(* CoDeSys 2.3 project: cy-wg-03_013.pro *)
(* Title: ClevergyAS - SanFelice *)
(* Version: 0.0 *)
(* Author: Andrea Ravasio *)
(* Libraries: serial_interface_01.lib 22.4.13 11:50:14, SerComm.lib 31.5.11 07:54:36, MBus_03.lib 9.2.13 16:51:58, Util.lib 18.5.10 14:14:28, Visual.lib 2.12.10 13:48:34, WagoLibIdent.lib 25.2.13 10:12:16, WagoLibStatus.lib 2.12.10 13:48:32, SysLibFile.lib 2.12.10 13:48:34, SysLibRtc.lib 2.12.10 13:48:32, SysLibSockets.lib 10.2.11 08:20:54, SysLibEvent.lib 2.12.10 13:48:34, SysLibPlcCtrl.lib 2.12.10 13:48:32, Standard.lib 2.12.10 13:48:34, SYSLIBCALLBACK.LIB 2.12.10 13:48:32 *)

(* PLC configuration (modules and I/O channels)
0750-0402 4 DI 24 V DC 3.0ms [Type_1_4_Channels] node 0, in %IB24 out %QB4 {INTTypePAAssignment = PLC; INTTypeModule = plugged}
  VPN_ST2 AT %IX12.0 [BOOLOnX_I] Ch_1 Digital input
  KEY_QE_ST AT %IX12.1 [BOOLOnX_I] Ch_2 Digital input
  AT %IX12.2 [BOOLOnX_I] Ch_3 Digital input
  PORT01_DI AT %IX12.3 [BOOLOnX_I] Ch_4 Digital input
0750-0402 4 DI 24 V DC 3.0ms [Type_1_4_Channels] node 1, in %IB24 out %QB4 {INTTypePAAssignment = PLC; INTTypeModule = plugged}
  GAS02_DI AT %IX12.4 [BOOLOnX_I] Ch_1 Digital input
  GAS01_DI AT %IX12.5 [BOOLOnX_I] Ch_2 Digital input
  AT %IX12.6 [BOOLOnX_I] Ch_3 Digital input
  AT %IX12.7 [BOOLOnX_I] Ch_4 Digital input
0750-0504 4 DO 24V DC 0.5A [Type_10_4_Channels] node 2, in %IX12.4 out %QB4 {INTTypePAAssignment = PLC; INTTypeModule = plugged}
  AT %QX2.0 [BOOLOnX_Q] Ch_1 Digital output
  AT %QX2.1 [BOOLOnX_Q] Ch_2 Digital output
  AT %QX2.2 [BOOLOnX_Q] Ch_3 Digital output
  AT %QX2.3 [BOOLOnX_Q] Ch_4 Digital output
0750-0504 4 DO 24V DC 0.5A [Type_10_4_Channels] node 3, in %IB25 out %QB4 {INTTypePAAssignment = PLC; INTTypeModule = plugged}
  AT %QX2.4 [BOOLOnX_Q] Ch_1 Digital output
  AT %QX2.5 [BOOLOnX_Q] Ch_2 Digital output
  TEST1 AT %QX2.6 [BOOLOnX_Q] Ch_3 Digital output
  TEST2 AT %QX2.7 [BOOLOnX_Q] Ch_4 Digital output
0750-0464#02 2/4 AI RTD / ADJ./ HA [Type_44_2_Channels] node 4, in %IB20 out %QB0 {INTTypePAAssignment = PLC; INTTypeModule = plugged}
  TT_S01 AT %IW0 [INTOnW_I] Ch_1 signed Input value
  AT %IW1 [INTOnW_I] Ch_2 signed Input value
0750-0472 2 AI 0-20mA 16 Bit S.E. [Type_8_2_Channels] node 5, in %IB20 out %QB0 {INTTypePAAssignment = PLC; INTTypeModule = plugged}
  TT_S07 AT %IW2 [WORDOnW_I] I 1: Analog Input
  TT_S06 AT %IW3 [WORDOnW_I] I 2: Analog Input
0750-0472 2 AI 0-20mA 16 Bit S.E. [Type_8_2_Channels] node 6, in %IB24 out %QB0 {INTTypePAAssignment = PLC; INTTypeModule = plugged}
  TT_S05 AT %IW4 [WORDOnW_I] I 1: Analog Input
  TT_S04 AT %IW5 [WORDOnW_I] I 2: Analog Input
0750-0472 2 AI 0-20mA 16 Bit S.E. [Type_8_2_Channels] node 7, in %IB28 out %QB0 {INTTypePAAssignment = PLC; INTTypeModule = plugged}
  TT_S03 AT %IW6 [WORDOnW_I] I 1: Analog Input
  TT_S02 AT %IW7 [WORDOnW_I] I 2: Analog Input
0750-0472 2 AI 0-20mA 16 Bit S.E. [Type_8_2_Channels] node 8, in %IB32 out %QB0 {INTTypePAAssignment = PLC; INTTypeModule = plugged}
  PORT01_AI AT %IW8 [WORDOnW_I] I 1: Analog Input
  AT %IW9 [WORDOnW_I] I 2: Analog Input
0750-0650/0003-0000#03 RS 232 C Interface (Adjustable), 3 Byte [Type_21_1_Channels] node 9, in %IB36 out %QB0 {INTTypePAAssignment = PLC; INTTypeModule = plugged}
  AT %IX10.0 [BOOLOnX_I] Transmission acknowledgement
  AT %IX10.1 [BOOLOnX_I] Reception request
  AT %IX10.2 [BOOLOnX_I] Initialization acknowledgement
  AT %IX10.3 [BOOLOnX_I] Input buffer is full
  AT %IX10.4 [BOOLOnX_I] Number of received characters Bit 0
  AT %IX10.5 [BOOLOnX_I] Number of received characters Bit 1
  AT %IX10.6 [BOOLOnX_I] Number of received characters Bit 2
  AT %IB21 [BYTEOnB_I] Input data Byte 0
  AT %IB22 [BYTEOnB_I] Input data Byte 1
  AT %IB23 [BYTEOnB_I] Input data Byte 2
  AT %QX0.0 [BOOLOnX_Q] Transmission request
  AT %QX0.1 [BOOLOnX_Q] Reception acknowledgement
  AT %QX0.2 [BOOLOnX_Q] Initialization request
  AT %QX0.4 [BOOLOnX_Q] Number of characters Bit 0
  AT %QX0.5 [BOOLOnX_Q] Number of characters Bit 1
  AT %QX0.6 [BOOLOnX_Q] Number of characters Bit 2
  AT %QB1 [BYTEOnB_Q] Output data Byte 0
  AT %QB2 [BYTEOnB_Q] Output data Byte 1
  AT %QB3 [BYTEOnB_Q] Output data Byte 2
Fieldbus variables [FB_VARS] node 1, in %IB0 out %QB0
Flag variables [FLAG_VARS] node 2, in %IB0 out %QB0
Modbus-Master [MB_MASTER] node 3, in %IB0 out %QB0
*)

(* Global variable list: Global_Constants *)
VAR_GLOBAL CONSTANT

	Plant_NAME			: STRING :='cySN:3 cyVER:14 - San Felice';
	Plant_SN			: DWORD :=3;   		(* S/N Impianto di telecontrollo *)
	Plant_SW_VER		: WORD  :=14;		(* Versione SW installata *)

	(* Parameters *)
	Plant_DefaultTAmb	: INT	:=100;		(* [.1°C] Temperatura ambiente di default in caso di rottura sonda *)

	(* Filesystem *)
	FilesPath  			: STRING :='S:\';

	(* TCP Logger *)
	Logger_SERVER		: STRING:='';
	Logger_IP			: STRING:='192.168.100.3';
	Logger_PORT			: WORD  :=80;
	Logger_GETSTART		: STRING:='GET /cygmsrv/hsgm.ashx?';
	Logger_GETEND		: STRING:='$R$N$R$N';
	Logger_CHECK		: STRING:='True';
	Logger_CRLF			: STRING:='$R$N';
	Logger_DataFile		: STRING:='S:\LOG.DAT';
	Logger_DataFileOld	: STRING:='S:\LOG.BCK';
	Logger_IndexFile	: STRING:='S:\LOG.IDX';
	Logger_ConnRetries	: BYTE:=5;
	Logger_RecoverMsgs	: BYTE:=100;

	(* TCP Remote *)
	Remote_PORT			: WORD  :=10;
	Remote_WELCOME		: STRING:='Connected$R$N';
	Remote_OK			: STRING:='OK$R$N';
	Remote_ERROR		: STRING:='ERROR$R$N';

	(* TCP Sockets *)
	MAX_SEND_TCP_SERVER					 : DWORD:=1500;(*60000*)
	MAX_RECEIVE_TCP_SERVER				 : DWORD:=3000;
	MAX_RECEIVE_TCP_SERVER_SOCKET	 	 : DWORD:=1500;
	MAX_SEND_TCP_CLIENT					 : DWORD:=1500;(*15000*)
	MAX_RECEIVE_TCP_CLIENT				 : DWORD:=1500;
	MAX_RECEIVE_TCP_CLIENT_SOCKET		 : DWORD:=1500;
	MAX_RECEIVE_UDP_SERVER				 : INT  :=1472;
	MAX_RECEIVE_UDP_CLIENT				 : INT  :=1472;
	CONNECT_WATCHDOG_TIME				 : TIME :=t#10s;

END_VAR

(* Global variable list: Global_Retain *)
VAR_GLOBAL RETAIN PERSISTENT

	PortataTotalePORT01		: DINT;
	ConteggioTotalePORT01	: DINT;
	PortataTotaleGAS01		: DINT;
	ConteggioTotaleGAS01	: DINT;
	PortataTotaleGAS02		: DINT;
	ConteggioTotaleGAS02	: DINT;

	CTB250_ENERGY_WH		: REAL;
	CTB250_ENERGY			: DWORD; (* 10^-2 MWh *)

	Mode_Manual : BOOL := FALSE;
END_VAR

(* Global variable list: Global_Variables *)
VAR_GLOBAL

	SYS    : typ_SYS;
	T_AMB  : INT;

	TPV01  : obj_TPV		:= ( ID:=1,
								 IN_EMIN:=-600 , IN_EMAX:=2500 ,
								 IN_WMIN:=-500 , IN_WMAX:=600 ); (* T_S01 *)

	TPV02  : obj_TPV_SENS	:= ( ID:=2 ,
											SogliaHL:=4096 ,   	 	(* Soglia Sonda Aperta = 2,5mA *)
											SogliaHH:=32767,	 	(* Soglia Sonda CC = 20mA *)
											SogliaWL:=10, 			(* Soglia WRN Bassa  = 10°C *)
											SogliaWH:=120,			(* Soglia WRN Alta  = 120°C *)
											PuntoMinX:=0, 		    (* Scalatura Minima vedi data di targa sonda 0°C *)
											PuntoMaxX:=160,			(* Scalatura Massima Vedi data di targa Sonda 160°C *)
											PuntoMinY:=6553,		(* Valore minimio per scalatura = 4mA *)
											PuntoMaxY:=32767,		(* Valore Massimo per Scalatura = 20mA *)
											Decimali:=1); 			(* Decimali da ottenere durante la scalatura *)
	TPV03  : obj_TPV_SENS	:= ( ID:=3 ,
											SogliaHL:=4096 ,   	 	(* Soglia Sonda Aperta = 2,5mA *)
											SogliaHH:=32767,	 	(* Soglia Sonda CC = 20mA *)
											SogliaWL:=10, 			(* Soglia WRN Bassa  = 10°C *)
											SogliaWH:=120,			(* Soglia WRN Alta  = 120°C *)
											PuntoMinX:=0, 		    (* Scalatura Minima vedi data di targa sonda 0°C *)
											PuntoMaxX:=160,			(* Scalatura Massima Vedi data di targa Sonda 160°C *)
											PuntoMinY:=6553,		(* Valore minimio per scalatura = 4mA *)
											PuntoMaxY:=32767,		(* Valore Massimo per Scalatura = 20mA *)
											Decimali:=1); 			(* Decimali da ottenere durante la scalatura *)

	TPV04  : obj_TPV_SENS	:= ( ID:=4 ,
											SogliaHL:=4096 ,   	 	(* Soglia Sonda Aperta = 2,5mA *)
											SogliaHH:=32767,	 	(* Soglia Sonda CC = 20mA *)
											SogliaWL:=10, 			(* Soglia WRN Bassa  = 10°C *)
											SogliaWH:=120,			(* Soglia WRN Alta  = 120°C *)
											PuntoMinX:=0, 		    (* Scalatura Minima vedi data di targa sonda 0°C *)
											PuntoMaxX:=160,			(* Scalatura Massima Vedi data di targa Sonda 160°C *)
											PuntoMinY:=6553,		(* Valore minimio per scalatura = 4mA *)
											PuntoMaxY:=32767,		(* Valore Massimo per Scalatura = 20mA *)
											Decimali:=1); 			(* Decimali da ottenere durante la scalatura *)

	TPV05  : obj_TPV_SENS	:= ( ID:=5 ,
											SogliaHL:=4096 ,   	 	(* Soglia Sonda Aperta = 2,5mA *)
											SogliaHH:=32767,	 	(* Soglia Sonda CC = 20mA *)
											SogliaWL:=10, 			(* Soglia WRN Bassa  = 10°C *)
											SogliaWH:=120,			(* Soglia WRN Alta  = 120°C *)
											PuntoMinX:=0, 		    (* Scalatura Minima vedi data di targa sonda 0°C *)
											PuntoMaxX:=160,			(* Scalatura Massima Vedi data di targa Sonda 160°C *)
											PuntoMinY:=6553,		(* Valore minimio per scalatura = 4mA *)
											PuntoMaxY:=32767,		(* Valore Massimo per Scalatura = 20mA *)
											Decimali:=1); 			(* Decimali da ottenere durante la scalatura *)

	TPV06  : obj_TPV_SENS	:= ( ID:=6 ,
											SogliaHL:=4096 ,   	 	(* Soglia Sonda Aperta = 2,5mA *)
											SogliaHH:=32767,	 	(* Soglia Sonda CC = 20mA *)
											SogliaWL:=10, 			(* Soglia WRN Bassa  = 10°C *)
											SogliaWH:=120,			(* Soglia WRN Alta  = 120°C *)
											PuntoMinX:=0, 		    (* Scalatura Minima vedi data di targa sonda 0°C *)
											PuntoMaxX:=160,			(* Scalatura Massima Vedi data di targa Sonda 160°C *)
											PuntoMinY:=6553,		(* Valore minimio per scalatura = 4mA *)
											PuntoMaxY:=32767,		(* Valore Massimo per Scalatura = 20mA *)
											Decimali:=1); 			(* Decimali da ottenere durante la scalatura *)

	TPV07  : obj_TPV_SENS	:= ( ID:=7 ,
											SogliaHL:=4096 ,   	 	(* Soglia Sonda Aperta = 2,5mA *)
											SogliaHH:=32767,	 	(* Soglia Sonda CC = 20mA *)
											SogliaWL:=10, 			(* Soglia WRN Bassa  = 10°C *)
											SogliaWH:=120,			(* Soglia WRN Alta  = 120°C *)
											PuntoMinX:=0, 		    (* Scalatura Minima vedi data di targa sonda 0°C *)
											PuntoMaxX:=160,			(* Scalatura Massima Vedi data di targa Sonda 160°C *)
											PuntoMinY:=6553,		(* Valore minimio per scalatura = 4mA *)
											PuntoMaxY:=32767,		(* Valore Massimo per Scalatura = 20mA *)
											Decimali:=1); 			(* Decimali da ottenere durante la scalatura *)
	(* Misuratore di Portata *)
	PORT01  : obj_PORT	:=  ( ID:=1 ,
											Peso:=1,				(* Peso del'impulso *)
											TempoTimeOut:=T#1m,		(* Minuti di attesa prima di segnalare WRN di inattività sulla linea *)
											SogliaHL:=4096,   	 	(* Soglia Sonda Aperta = 2,5mA *)
											SogliaHH:=32767,	 	(* Soglia Sonda CC = 20mA *)
											SogliaWL:=100, 			(* Soglia WRN Bassa  = ##### m3/h *)
											SogliaWH:=700,			(* Soglia WRN Alta  = ##### m3/h *)
											PuntoMinX:=0, 		    (* Scalatura Minima vedi data di targa sonda ##### m3/h *)
											PuntoMaxX:=800,			(* Scalatura Massima Vedi data di targa Sonda  ##### m3/h *)
											PuntoMinY:=6553,		(* Valore minimio per scalatura = 4mA *)
											PuntoMaxY:=32767,		(* Valore Massimo per Scalatura = 20mA *)
											Decimali:=0); 			(* Decimali da ottenere durante la scalatura *)

	(*  Contatori *)
	GAS01  : obj_GAS:=  (ID:=1,	Peso:=33 ,				(* Peso del'impulso *)
								TempoTimeOut:=T#1m		(* Minuti di attesa prima di segnalare WRN di inattività sulla linea *)
													  );
	GAS02  : obj_GAS:=  (ID:=2,	Peso:=77 ,				(* Peso del'impulso *)
								TempoTimeOut:=T#1m		(* Minuti di attesa prima di segnalare WRN di inattività sulla linea *)
													  );

	(* Contabilizzatori *)
	MBUS01 	  : obj_MBUS				:= ( ID:=1 , COM:=2 , BAUDRATE:=BAUD_2400 );
	CTBSCAN01 : obj_MBUS_CTB_SCANNER	:= ( ID:=1 );
	CTB250	  : obj_SW_CTB				:= ( ID:=250 );

	Logger : typ_Logger;

	(**** SIMULATION ONLY ****)
	(*...*)
END_VAR

(* Data type in Errors *)
TYPE en_Logger_ErrLev :
(
	EL_Log			:=0,
	EL_Wrn			:=1,
	EL_Alarm		:=2,
	EL_AlarmStop	:=3
);
END_TYPE

(* Data type in Errors *)
TYPE en_Logger_Status :
(
	S_Logger_UNKNOWN := 0,
	S_Logger_IDLE,
	S_Logger_WAITCONN,
	S_Logger_WAITTX,
	S_Logger_WAITRESP,
	S_Logger_ERROR
);
END_TYPE

(* Data type *)
TYPE en_SYS_Objects :
(
	EO_SYS		:=0,  (* PLC *)
	EO_VPN		:=1,  (* VPN *)
	EO_DOOR		:=2,  (* Door & access control *)

	EO_CAL		:=10, (* Caldaia *)
	EO_CIR		:=11, (* Circolatore *)
	EO_CRON		:=12, (* Crono-termostato *)
	EO_VRD		:=13, (* Valvola miscelatore pannelli *)
	EO_CTL		:=14, (* Contalitri *)
	EO_CTB		:=15, (* Contabilizzatore *)
	EO_TPV		:=16, (* Temperature probes values *)
	EO_PPV		:=17, (* Pressure probes values *)
	EO_PBV		:=18, (* Over-Pressure Alarms *)
	EO_TBV		:=19, (* Over-Temperature Alarms *)
	EO_PMV		:=20, (* Under-Pressure Alarms *)
	EO_GRU		:=21, (* Gruppo termico *)
	EO_PDC		:=22, (* Pompa di calore *)
	EO_SOL		:=23, (* Pannello solare termico *)
	EO_ESOL		:=24, (* Pannello solare fotovoltaico *)
	EO_GAS		:=25, (* Contatore GAS *)
	EO_PORT		:=26, (* Misuratore di portata *)
	EO_FPV		:=27, (* Flow probes values *)

	EO_LON		:=1000, (* Bus - LON *)
	EO_MODBUS	:=1001, (* Bus - MODBUS *)
	EO_MBUS		:=1002  (* Bus - M-BUS *)
);
END_TYPE

(* Data type *)
TYPE en_SYS_Status :
(
	S_UNKNOWN  := 0,
	S_STARTUP,
	S_INIT_RTC,
	S_INIT_VAR,
	S_AUTOTEST,
	S_RUNNING,
	S_SHUTDOWN,
	S_HALT
);
END_TYPE

(* Data type in Errors *)
TYPE typ_Logger :
STRUCT
	Status		: en_Logger_Status;

	SendReq		: BOOL;
	SendIdx		: DWORD;
	SendData	: ARRAY [0..MAX_SEND_TCP_CLIENT] OF BYTE;
	SendLen		: DINT;

	TData		: ARRAY [0..MAX_SEND_TCP_CLIENT] OF BYTE;
	TLen		: DINT;

	LastIdxPos	: DWORD;

END_STRUCT
END_TYPE

(* Data type *)
TYPE typ_SYS :
STRUCT
	Status			: en_SYS_Status;
	Warning			: BOOL;
	Alarm			: BOOL;
	AlarmStop		: BOOL;

	Time_LogString	: STRING;
	Time_Year		: WORD;
	Time_Month		: BYTE;
	Time_Day		: BYTE;

	Time_CT_DT		: DT;
	Time_CT_Day		: WORD;
	Time_CT_Quarter	: BYTE;

	LastLogs_Idx	: BYTE;
	LastLogs_Dat	: ARRAY[0..5] OF STRING;
	LastLogs_Msg	: ARRAY[0..5] OF STRING;

END_STRUCT
END_TYPE

(* Data type in Plant_Objects *)
TYPE typ_VisuStrutturaMbus :
STRUCT

	sdNodoPresente: STRING(16);
	sdEnergia: STRING(16);
	sdPotenza: STRING(16);
	sdVolume: STRING(16);
	sdFlow: STRING(16);
	sdTempIngresso: STRING(8);
	sdTempaUscita: STRING(8);
	sdTempDelta: STRING(8);

END_STRUCT
END_TYPE

(* POU PLC_PRG, ST *)
PROGRAM PLC_PRG
VAR
	Timer1: TON; (* Fast controls tick *)
	Timer2: TON; (* Plant control tick *)
	Timer3: TON; (* Logger timer *)
END_VAR
(******************************************************************************
 ****                           MAIN TASK CODE                             ****
 ******************************************************************************

	Network setup:
		IP  = 192.168.100.2 | MSK = 255.255.255.0 | GW = 192.168.100.1
		DNS = 192.168.100.1 | NTP = 193.168.100.3

	Editor setup:
		Project --> Options --> Editor --> Fonts --> Courier NEW / BOLD / 12

*)

(*==============================*)
(*===== Main status machine ====*)
(*==============================*)
Main_Stm();

(*=====================================*)
(*== Running common cycle operations ==*)
(*=====================================*)
IF SYS.Status>S_INIT_VAR THEN

	(* Execute M-BUS processes *)
	MBUS01();
	CTBSCAN01( MBUS:=MBUS01 );

END_IF


(*==============================*)
(*== System cycle operations ===*)
(*==============================*)
(* Execute TCP processes *)
Logger_Proc();
Remote_Proc();
(* Update user led *)
USRLED_Update();
(* Execute Cron Editor commands *)
(*...*)
(* External resources *)
IF TPV01.ERR THEN T_AMB:=Plant_DefaultTAmb; ELSE T_AMB:=TT_S01; END_IF

(**** SIMULATION ONLY ****)
(*...*)
END_PROGRAM
ACTION Main_Stm:
CASE Sys.Status OF
	(*--------------------------------------------------------*)
	S_STARTUP:
		Sys.Status:=S_INIT_RTC;
	(*--------------------------------------------------------*)
	S_INIT_RTC:
		(* Check RTC and update from network *)
		RTC_Update();
		(* Check time *)
		IF Sys.Time_Year>2000 THEN
			Sys.Status:=S_INIT_VAR;
		END_IF
	(*--------------------------------------------------------*)
	S_INIT_VAR:
		LogEv(EL_Wrn,EO_SYS,0,1,CONCAT('System_startup_v',WORD_TO_STRING(Plant_SW_VER)));
		Sys.Status:=S_RUNNING;
	(*--------------------------------------------------------*)
	S_RUNNING:

		Timer1(IN:=NOT Timer1.Q,PT:=T#50ms);
		IF Timer1.Q THEN
			(* Update system checks *)
			SYS_Proc();
		END_IF

		Timer2(IN:=NOT Timer2.Q,PT:=T#500ms);
		IF Timer2.Q THEN
			(* Read current date/time *)
			RTC_Update();
			(* === Execute plant operations === *)
			(* Temperature da RTD *)
			TPV01	 ( IN:=TT_S01 );
			(* Temperature da Convertitori 4-20mA *)
			TPV02	 ( AI_INPUT:=TT_S02 );
			TPV03	 ( AI_INPUT:=TT_S03 );
			TPV04	 ( AI_INPUT:=TT_S04 );
			TPV05	 ( AI_INPUT:=TT_S05 );
			TPV06	 ( AI_INPUT:=TT_S06 );
			TPV07	 ( AI_INPUT:=TT_S07 );
			(* Contabilizzatori Digitali *)
			CTB250   (	T_SEND:=(TPV02.ValoreScalato+TPV03.ValoreScalato+TPV04.ValoreScalato)/3,
						T_RET :=(TPV05.ValoreScalato+TPV06.ValoreScalato+TPV07.ValoreScalato)/3,
						FLOW  :=PORT01.ValoreScalato,
						ENERGY_WH:=CTB250_ENERGY_WH,
						ENERGY   :=CTB250_ENERGY );

			(* Test toggle *)
			IF TEST1 THEN TEST1:=FALSE; ELSE TEST1:=TRUE; END_IF
		     END_IF

		Timer3(IN:=NOT Timer3.Q,PT:=T#5m);
		IF Timer3.Q THEN
			(* Trig logger *)
			LogTrig();
			(* Execute temporary CSV logger *)
			CSV_Log();
		END_IF

		(* Contabilizzatori Digitali *)
		PORT01( DI_Input:=PORT01_DI, AI_INPUT:=PORT01_AI,
				Totalizzatore:=PortataTotalePORT01,
				Contatore:=ConteggioTotalePORT01 );
		GAS01 ( DI_Input:=GAS01_DI,
				Totalizzatore:=PortataTotaleGAS01,
				Contatore:=ConteggioTotaleGAS01 );
		GAS02 ( DI_Input:=GAS02_DI,
				Totalizzatore:=PortataTotaleGAS02,
				Contatore:=ConteggioTotaleGAS02 );

	(*--------------------------------------------------------*)
	S_SHUTDOWN:
		(* Arresto del sistema *)
		Sys.Status:=S_STARTUP;
	(*--------------------------------------------------------*)
	S_HALT:
		(* Aspetta uscita manuale *)
		Sys.Status:=S_STARTUP;
	(*--------------------------------------------------------*)
ELSE
	Sys.Status:=S_STARTUP;
END_CASE;
END_ACTION

(* POU TCP_Logger/Logger_Proc, ST *)
PROGRAM Logger_Proc
VAR
	c1:         	TCPCLIENT;

	Open:	    	BOOL;
	IpAddr:			DWORD;
	InetAddr:		DWORD;
	Connected:  	BOOL;
	Error:      	DINT;
	TxTrig:     	BOOL;
	RxData:			ARRAY [0..MAX_RECEIVE_TCP_CLIENT] OF BYTE;
	RxLen:			DINT;

	Retry:			BYTE;	(* Counter for connection retries *)
	Recovered:		BYTE;	(* Counter for recovered unsent messages *)

	i:				DINT;
	pos:			DWORD;
	hFile:			DWORD;

END_VAR
(*=== State machine ===*)
CASE Logger.Status OF

	S_Logger_UNKNOWN:
		(* Startup *)
		Logger.SendReq:=FALSE;
		Open:=FALSE;
		Logger.Status:=S_Logger_IDLE;

	S_Logger_IDLE:
		(* Wait request *)
		IF Logger.SendReq THEN
			(* Resolve server name or use static IP *)
			IF LEN(Logger_SERVER)=0 THEN
				InetAddr:=SysSockInetAddr(Logger_IP);
			ELSE
				IpAddr:=SysSockGetHostByName(ADR(Logger_SERVER));
				DWORDSWAP(pIn:=ADR(IpAddr), pOut:=ADR(InetAddr));
			END_IF
			TxTrig:=FALSE;
			RxLen:=0;
			(* Open connection *)
			Open:=TRUE;
			Logger.Status:=S_Logger_WAITCONN;
		END_IF

	S_Logger_WAITCONN:
		(* Wait connection *)
		IF Connected THEN
			(* Send data *)
			TxTrig:=TRUE;
			Logger.Status:=S_Logger_WAITTX;
		END_IF
		IF Error>0 THEN
			Open:=FALSE;
			Logger.Status:=S_Logger_ERROR;
		END_IF

	S_Logger_WAITTX:
		(* Wait transmission *)
		IF NOT TxTrig THEN
			Logger.Status:=S_Logger_WAITRESP;
		END_IF
		IF Error>0 THEN
			Open:=FALSE;
			Logger.Status:=S_Logger_ERROR;
		END_IF

	S_Logger_WAITRESP:
		(* Wait response *)
		IF Connected=FALSE (* OR TIMEOUT!! *) THEN
			Open:=FALSE;
			(* Check response *)
			IF RxLen>=4 AND CHKSTRING(pString:=ADR(RxData), pPattern:=ADR(Logger_CHECK)) THEN
				Logger.SendReq:=FALSE;
				Retry:=0;
				(* Check unsent messages to flush *)
				IF Recovered<Logger_RecoverMsgs THEN
					MsgChk();
					IF Logger.SendReq=TRUE THEN
						Recovered:=Recovered+1;
					ELSE
						Recovered:=0;
					END_IF
				ELSE
					Recovered:=0;
				END_IF
				Logger.Status:=S_Logger_IDLE;
			ELSE
				Logger.Status:=S_Logger_ERROR;
			END_IF
		END_IF

	S_Logger_ERROR:
		(* Connection error or send failure *)
		Retry:=Retry+1;
		IF Retry>Logger_ConnRetries THEN
			(* Save message as unsent *)
			MsgSave();
			Logger.SendReq:=FALSE;
			Retry:=0;
		END_IF
		Logger.Status:=S_Logger_IDLE;

ELSE
	Logger.Status:=S_Logger_UNKNOWN;
END_CASE


(*=== Execute client lib ===*)
c1(
	xOpenConnection			:= Open,
	dwInetAddr 				:= InetAddr,
	wPortNumber				:= Logger_PORT,
	ptSendData				:= ADR(Logger.SendData),
	diSendCount				:= Logger.SendLen,
	tConnectWatchdogTime	:= t#10s,
	xStartSend				:= TxTrig,
	aReceiveBuffer			:= RxData,
	diReceiveCount			:= RxLen,
	xConnected				=> Connected,
	diError					=> Error
);

(*=== Process Rx data ===*)
(*IF RxLen>0 THEN
	RxLen:=0;
END_IF*)
END_PROGRAM
ACTION MsgChk:
(* Open index file *)
hFile:=SysFileOpen(Logger_IndexFile,'r');
IF hFile=0 THEN
	RETURN;
END_IF
(* Search oldest message to recover *)
SysFileSetPos(hFile,Logger.LastIdxPos);
Logger.SendLen:=0;
REPEAT
	SysFileRead(hFile, ADR(Logger.SendIdx), SIZEOF(Logger.SendIdx));
	pos:=SysFileGetPos(hFile);
	SysFileRead(hFile, ADR(Logger.SendLen), SIZEOF(Logger.SendLen));
UNTIL
	SysFileEOF(hFile) OR Logger.SendLen<>0
END_REPEAT
SysFileClose(hFile);
(* Delete index file when all messages are recovered *)
IF Logger.SendLen=0 THEN
	Logger.LastIdxPos:=0;
	SysFileDelete(Logger_IndexFile);
	RETURN;
END_IF
(* Recover message data *)
hFile:=SysFileOpen(Logger_DataFile,'r');
IF hFile<>0 THEN
	SysFileSetPos(hFile,Logger.SendIdx);
	SysFileRead(hFile,ADR(Logger.SendData),Logger.SendLen);
	Logger.SendReq:=TRUE;
	SysFileClose(hFile);
END_IF
(* Clear index entry *)
hFile:=SysFileOpen(Logger_IndexFile,'a');
IF hFile<>0 THEN
	SysFileSetPos(hFile,pos);
	i:=0;
	SysFileWrite(hFile, ADR(i), 4);
	Logger.LastIdxPos:=SysFileGetPos(hFile);
	SysFileClose(hFile);
END_IF
END_ACTION
ACTION MsgSave:
(* Add log position in recovery indexes *)
hFile:=SysFileOpen(Logger_IndexFile,'a');
SysFileWrite(hFile, ADR(Logger.SendIdx), SIZEOF(Logger.SendIdx));
SysFileWrite(hFile, ADR(Logger.SendLen), SIZEOF(Logger.SendLen));
SysFileClose(hFile);
END_ACTION

(* POU Utils Functions/TCPCLIENT, ST *)
FUNCTION_BLOCK TCPCLIENT
(***********************************************************************************************************	*)
(* Version: 1.3b                        			          													*)
(* Date: 28.10.2014                   				          							            			*)
(***********************************************************************************************************	*)
(* WAGO Kontakttechnik GmbH Hansastr. 27 32423 Minden(Westf.)													*)
(* Tel. +0049 571/887-0 Fax. +0049 571/887-0																	*)
(* Author: VB																									*)
(***********************************************************************************************************	*)
(*Description:	A TCP client to read and write data with additional connection watchdog							*)
(*History:																										*)
(*Version 1.3b: 28.10.2014: Use DWORD address for IP (Andrea Ravasio)											*)
(*Version 1.3: 11.02.2011: Changes according to 750-880/881											 			*)
(*Version 1.2: 29.08.2007 Bugfix TCP Client																		*)
(*Version 1.1: 15.01.2007 Changes according to FW11																*)
(*Version 1.0: 09.03.2006 Release																				*)
(***********************************************************************************************************	*)
VAR CONSTANT
	STATE_CREATE     				 : BYTE:= 0;
	STATE_OPEN     					 : BYTE:= 1;
	STATE_IOCTL    					 : BYTE:= 2;
	STATE_CONNECT     				 : BYTE:= 10;
	STATE_TX       					 : BYTE:= 20;
	STATE_RX       					 : BYTE:= 30;
	STATE_CLOSE    					 : BYTE:= 40;
	STATE_ERROR_TRAP			     : BYTE:= 200;
END_VAR

VAR_INPUT
	xOpenConnection					: BOOL;
	dwInetAddr						: DWORD; (* <== Use SysSockInetAddr() value or
													swapped bytes order of SysSockGetHostByName() value *)
	wPortNumber						: WORD;
	ptSendData						: POINTER TO ARRAY[0..MAX_SEND_TCP_CLIENT] OF BYTE;
	diSendCount						: DINT;
	tConnectWatchdogTime		    : TIME := t#10s;
END_VAR
VAR_OUTPUT
	xConnected						: BOOL;
	diError 						: DINT := 0;
END_VAR
(* ErrorCodes -----------------------------------------
	16#8001 => No socket descriptor available 
	16#8002 => SysSockSend returns -1 
	16#8003 => Socket was "gracefully closed" 
	16#8004 => switching to none blocking mode fails
	16#8005 => SysSockClose() returns FALSE 
    16#8006 => SysSockConnect() fails
    16#8007 => SysSockSend() fails
	16#8008 => error state machine 
	16#8009 => timeout while waiting for data from server 
------------------------------------------------------------*)
VAR_IN_OUT
	xStartSend							: BOOL;
	aReceiveBuffer						: ARRAY [0..MAX_RECEIVE_TCP_CLIENT] OF BYTE;
	diReceiveCount						: DINT;
END_VAR
VAR
	m_State								: BYTE := 0;
	m_ReceiveBuffer						: ARRAY [0..MAX_RECEIVE_TCP_CLIENT_SOCKET] OF BYTE;
	m_Socket							: DINT;
	m_AddressInfo						: SOCKADDRESS;
	m_BytesReceived						: DINT;
	m_diReturn							: DINT;
	m_xReturn							: BOOL;
	m_IoCtlParameter  					: DINT := 1; (* IOCTL-Parameter for non-blocking mode of sockets *)
	i									: INT;
	T_Connect							: TON;
	m_count								: DINT;
	diOption							: DINT := 1;
	m_Blocking   						: DINT := 0;
END_VAR
IF xOpenConnection THEN
	(* State maschine *)
	CASE  m_State OF

	(* -------------------------------------------------------------------------*)
	STATE_CREATE:
			(* create socket descriptor*)
			m_Socket := SysSockCreate(diAddressFamily	:= SOCKET_AF_INET,
													 diType		:= SOCKET_STREAM,
													 diProtocol := SOCKET_IPPROTO_TCP);
			IF m_Socket >= 0 THEN
			(*Set Push-Bit*)
				IF ADR(%MW0)=16#30000000  OR ADR(%MW0)=16#20000000 THEN (*841 or 881*)
					SysSockSetOption(
						diSocket:=m_Socket,
						diLevel:=6,
						diOption:=SOCKET_TCP_NODELAY,
						pOptionValue:=ADR(diOption),
						diOptionLength:=SIZEOF(diOption));
				ELSE
						;
				END_IF
				m_State := STATE_IOCTL; (* succesful *)
			ELSE
				diError := 16#8001;  (* no socket descriptor available *)
				m_State := STATE_ERROR_TRAP;
			END_IF

	(* -------------------------------------------------------------------------*)
	STATE_IOCTL: (* change  socket mode  to none blocking *)
		m_diReturn := SysSockIoctl( m_Socket, SOCKET_FIONBIO, ADR(m_IoCtlParameter));
		IF m_diReturn <> 0 THEN
			m_AddressInfo.sin_family := SOCKET_AF_INET;
			m_AddressInfo.sin_port := SysSockNtohs(wPortNumber);
			m_AddressInfo.sin_addr := dwInetAddr;
			m_State := STATE_CONNECT;
		ELSE
			diError := 16#8004;  (* switching to none blocking mode fails *)
			m_State := STATE_ERROR_TRAP;
		END_IF


	(* -------------------------------------------------------------------------*)
	STATE_CONNECT: (* connect with server *)
		T_Connect(IN:=TRUE , PT:=tConnectWatchdogTime);(*activate watchdog for establishing connection to a server*)
		m_xReturn := SysSockConnect ( m_Socket, ADR(m_AddressInfo),  SIZEOF(m_AddressInfo));
		IF m_xReturn THEN (* succesful *)
			IF xStartSend THEN
				m_State := STATE_TX;(*transmit data*)
			ELSE
				m_State := STATE_RX;(*wait for data from server*)
			END_IF
			xConnected:=TRUE;
			T_Connect(IN:=FALSE);
		ELSE
			IF T_Connect.Q THEN
				diError := 16#8006;  (* connect fails *)
				xConnected:=FALSE;
				T_Connect(IN:=FALSE);
				m_State := STATE_ERROR_TRAP;
				SysSockClose( m_Socket);
			ELSE
				m_State := STATE_CONNECT;(*client still  tries to set up connection*)
			END_IF
		END_IF


	STATE_TX:	 (* send TCP-message *)
		m_diReturn := SysSockSend(diSocket := m_Socket,
								  pbyBuffer := ADR(ptSendData^[0]),
								  diBufferSize := diSendCount-m_count,
								  diFlags := 0);

		CASE m_diReturn OF
		-1:	(* ERROR *)
			T_Connect(IN:=TRUE , PT:=CONNECT_WATCHDOG_TIME);(*activate watchdog to check communication*)
			IF t_Connect.Q THEN
				diError := 16#8007;
				T_Connect(IN:=FALSE);
				m_State:=STATE_CLOSE;
			END_IF
		0: (* socket was "gracefully closed" *)
			m_State := STATE_CLOSE;
			diError := 16#8003;
		ELSE (* succesful *)
			m_count:=m_count+m_diReturn;
			IF m_count>=diSendCount THEN
				diError := 16#0000;
				m_State := STATE_RX;
				m_count:=0;
				xStartSend:=FALSE;
			END_IF
			T_Connect(IN:=FALSE);
		END_CASE

	(* -------------------------------------------------------------------------*)
	STATE_RX: (* process receive data *)
			m_BytesReceived := SysSockRecv(	diSocket 	:= m_Socket,
										pbyBuffer 	:= ADR(m_ReceiveBuffer),		(* Address of receive buffer *)
										diBufferSize:= SIZEOF(m_ReceiveBuffer),
										diFlags		:= 0);

			CASE m_BytesReceived OF
			-1:	(* No data available or error occured *)
				T_Connect(IN:=TRUE , PT:=tConnectWatchdogTime);(*activate watchdog to check communication*)
				IF t_Connect.Q THEN
					diError:=16#8009;
					T_Connect(IN:=FALSE);
					m_State:=STATE_CLOSE;
				END_IF
				IF xStartSend THEN
					m_State:=STATE_TX	;(* WAIT IN THIS STATE  and check for arriving data or new send command*)
				END_IF;
			0: (* socket was "gracefully closed"  *)
				m_State:=STATE_CLOSE;
				diError := 16#8003;
			ELSE (* succesful *)
				diError := 16#0000;
				T_Connect(IN:=FALSE);
				(* Copy received data into receive buffer *)
				FOR i:= 0 TO DINT_TO_INT(m_BytesReceived	)-1 DO
					aReceiveBuffer[diReceiveCount]:= m_ReceiveBuffer[i];
					diReceiveCount:=(diReceiveCount+1) MOD SIZEOF(aReceiveBuffer);
				END_FOR

			END_CASE

	(* -------------------------------------------------------------------------*)
	STATE_CLOSE : (* close socket *)
		IF ADR(%MW0)=16#30000000  OR ADR(%MW0)=16#20000000 THEN (*841 or 881*)
			;
		ELSE
			SysSockShutdown(m_Socket, 0);;(*870*)
		END_IF
		m_xReturn := SysSockClose( m_Socket);
		m_Socket := -1;
		m_State := 0; (* succesful *)
		xConnected:=FALSE;
		T_Connect(IN:=FALSE);
	(* -------------------------------------------------------------------------*)
	STATE_ERROR_TRAP: (* error handling *)
		xConnected:=FALSE;

	ELSE  (* Bad FSM code trap  *)
			m_State:= STATE_ERROR_TRAP;
			diError:= 16#8008;
	END_CASE

ELSE(*close connection*)
	IF m_Socket >= 0 THEN
		IF ADR(%MW0)=16#30000000  OR ADR(%MW0)=16#20000000 THEN (*841 or 881*)
			;
		ELSE
			SysSockShutdown(m_Socket, 0);;(*870*)
		END_IF
		SysSockClose( m_Socket);
	END_IF
	m_Socket := -1;
	diError := 16#0000;
	m_State := STATE_CREATE;
	xConnected:=FALSE;
	T_Connect(IN:=FALSE);
END_IF
END_FUNCTION_BLOCK

(* POU Utils Functions/DWORDSWAP, ST *)
FUNCTION DWORDSWAP:BOOL
VAR_INPUT
	pIn:POINTER TO ARRAY[1..4] OF BYTE;
	pOut:POINTER TO ARRAY[1..4] OF BYTE;
END_VAR
VAR
END_VAR
pOut^[1]:=pIn^[4];
pOut^[2]:=pIn^[3];
pOut^[3]:=pIn^[2];
pOut^[4]:=pIn^[1];
END_FUNCTION

(* POU Utils Functions/CHKSTRING, ST *)
FUNCTION CHKSTRING : BOOL
VAR_INPUT
	pString: POINTER TO BYTE;
	pPattern: POINTER TO BYTE;
END_VAR
VAR
END_VAR
CHKSTRING:=TRUE;
WHILE pPattern^<>0 AND CHKSTRING DO
	IF pPattern^<>pString^ THEN CHKSTRING:=FALSE; END_IF
	pString:=pString+1;
	pPattern:=pPattern+1;
END_WHILE
END_FUNCTION

(* POU TCP_Remote/Remote_Proc, ST *)
PROGRAM Remote_Proc
VAR
	s1:         	TCPSERVER;
	Enable: 		BOOL;
	Connected: 		BOOL;
	Error: 			DINT;

	TxData:			ARRAY[0..MAX_SEND_TCP_SERVER] OF BYTE;
	TxLen:			DINT;
	TxTrig:			BOOL;

	RxData:			ARRAY [0..MAX_RECEIVE_TCP_SERVER] OF BYTE;
	RxLen:			DINT;

	Status:			DINT;

	(* Command interpreter *)

	Cmd_Buf:		ARRAY [0..MAX_RECEIVE_TCP_SERVER] OF BYTE;
	Cmd_Buf_U16:	POINTER TO WORD;
	Cmd_Buf_INT:	POINTER TO INT;
	Cmd_BufLen:		WORD;
	Cmd_St:			WORD;

	Cmd_Obj:		WORD;
	Cmd_ObjIdx:		WORD;
	Cmd_C:			WORD;
	Cmd_R:			WORD;
	Cmd_CLen:		WORD;
	Cmd_RLen:		WORD;

	i : WORD;
	j : INT;

END_VAR
(*=== State machine ===*)
CASE Status OF
	0: (* Startup *)
		TxLen:=0; TxTrig:=FALSE;
		RxLen:=0;
		Enable:=TRUE;
		Status:=1;

	1: (* Wait incoming connection *)
		IF Connected THEN
			(* Send welcome message *)
			ADDSTRING(pTxData:=ADR(TxData), pString:=ADR(Remote_WELCOME), TxLen:=TxLen);
			TxTrig:=TRUE;
			Cmd_BufLen:=0;
			Cmd_St:=0;
			Status:=2;
		END_IF
		IF Error>1 THEN
			Enable:=FALSE;
			Status:=0;
		END_IF

	2: (* Wait command *)
		IF RxLen>0 THEN
			(*=== Interpreter start ===*)
			IF Cmd_BufLen+(RxLen/2)>=MAX_RECEIVE_TCP_SERVER THEN
				(* ERROR *)
				Cmd_BufLen:=0;
			ELSE
				i:=HEXTORAW(pString:=ADR(RxData), StringLen:=DINT_TO_WORD(RxLen), pData:=ADR(Cmd_Buf[Cmd_BufLen]));
				Cmd_BufLen:=Cmd_BufLen+i;
			END_IF
			IF Cmd_BufLen>=8 THEN
				Cmd_Buf_U16:=ADR(Cmd_Buf[6]);
				IF Cmd_BufLen>=(8+Cmd_Buf_U16^) THEN
					Cmd_CLen:=Cmd_Buf_U16^;
					Cmd_Buf_U16:=ADR(Cmd_Buf[0]); Cmd_Obj:=Cmd_Buf_U16^;
					Cmd_Buf_U16:=ADR(Cmd_Buf[2]); Cmd_ObjIdx:=Cmd_Buf_U16^;
					Cmd_Buf_U16:=ADR(Cmd_Buf[4]); Cmd_C:=Cmd_Buf_U16^;
					Command();
					Cmd_BufLen:=0;
				END_IF
			END_IF

			(*=== Interpreter end ===*)
			RxLen:=0;
		END_IF
		IF NOT Connected THEN
			Status:=1;
		END_IF

ELSE
	Status:=0;
END_CASE


(*=== Execute server lib ===*)
s1(
	xEnable				:= Enable,
	wPortNumber			:= Remote_PORT,
	tServerTimeOut		:= t#15m,
	ptSendData			:= ADR(TxData),
	diSendCount			:= TxLen,
	xStartSend			:= TxTrig,
	aReceiveBuffer		:= RxData,
	diReceiveCount		:= RxLen,
	xClientConnected	=> Connected,
	diError				=> Error
);
END_PROGRAM
ACTION Cmd_CTB:
(* Check index *)
IF Cmd_ObjIdx<>1 THEN
	Cmd_R:=2;
	RETURN;
END_IF

(* Process command *)
CASE Cmd_C OF

	1: (* START SCANNING *)
		CTBSCAN01.Refresh:=TRUE;

ELSE
	Cmd_R:=3;
END_CASE
END_ACTION
ACTION Cmd_SYS:
(* Check index *)
IF Cmd_ObjIdx<>0 THEN
	Cmd_R:=2;
	RETURN;
END_IF

(* Process command *)
CASE Cmd_C OF

	0: (* ECHO *)
		IF Cmd_CLen<>0 THEN
			TxLen:=0;
		END_IF

	1: (* LOG REQUEST *)
		LogTrig();

	2: (* REARM *)
		Sys.Warning:=FALSE;
		Sys.Alarm:=FALSE;
		Sys.AlarmStop:=FALSE;

ELSE
	Cmd_R:=3;
END_CASE
END_ACTION
ACTION Command:
(* Default response OK/NODATA *)
Cmd_R:=0;
Cmd_RLen:=0;
TxLen:=16;

(* Check object *)
CASE Cmd_Obj OF

	EO_SYS:
		Cmd_SYS();

	EO_CTB:
		Cmd_CTB();

ELSE
	Cmd_R:=1;
END_CASE

(* Generate response *)
IF TxLen>0 THEN
	RAWTOHEX(ADR(Cmd_Obj)	,2,ADR(TxData[ 0]));
	RAWTOHEX(ADR(Cmd_ObjIdx),2,ADR(TxData[ 4]));
	RAWTOHEX(ADR(Cmd_R)		,2,ADR(TxData[ 8]));
	RAWTOHEX(ADR(Cmd_RLen)	,2,ADR(TxData[12]));
	TxTrig:=TRUE;
END_IF
END_ACTION

(* POU Utils Functions/TCPSERVER, ST *)
FUNCTION_BLOCK TCPSERVER
(***********************************************************************************************************	*)
(* Version: 1.6                                    			          											*)
(* Date: 11.02.2011                                   					          							    *)
(***********************************************************************************************************	*)
(* WAGO Kontakttechnik GmbH Hansastr. 27 32423 Minden(Westf.)													*)
(* Tel. +0049 571/887-0 Fax. +0049 571/887-0																	*)
(* Author: VB																									*)
(***********************************************************************************************************	*)
(*Description:	A TCP server to read and write data													       		*)
(*Historie:																										*)
(*Version 1.6: 11.02.2011: Changes according to 750-880/881											 			*)
(*Version 1.5: 27.11.2008 Bugfix allow reuse port																*)
(*Version 1.4: 13.10.2008 Bugfix transmitting large data														*)
(*Version 1.3: 15.01.2007 Changes according to FW11																*)
(*Version 1.2: 09.03.2006 Changes for socket handle 0											       			*)
(*Version 1.1: 14.02.2005 Release																				*)
(***********************************************************************************************************	*)
VAR CONSTANT
	STATE_INIT     				 : BYTE:= 0;
	STATE_OPEN     				 : BYTE:= 1;
	STATE_TX       				 : BYTE:= 20;
	STATE_RX       				 : BYTE:= 30;
	STATE_CLOSE    				 : BYTE:= 40;
	STATE_ERROR_TRAP		 	 : BYTE:= 200;
END_VAR
VAR_INPUT
	xEnable    					: BOOL;	 (* Set TRUE to enable function block *)
	wPortNumber					: WORD;  (* Port *)
	tServerTimeOut				: TIME:=t#50s;
	ptSendData					: POINTER TO ARRAY[0..MAX_SEND_TCP_SERVER] OF BYTE;
	diSendCount					: DINT;
END_VAR
VAR_OUTPUT
	xClientConnected  			: BOOL:= FALSE;
	diError 					: DINT:= 0;
END_VAR
(* Status Codes -----------------------------------------
	16#8001 => No socket descriptor available 
	16#8002 => SysSockBind fails 
	16#8003 => SysSockListen fails 
	16#8004 => switching to none blocking mode fails
	16#8005 => SysSockClose() returns FALSE 
    16#8006 => SysSockConnect() fails
    16#8007 => SysSockSend() fails
	16#8008 => error state machine 
	16#8009 => timeout while waiting for data from server 
	16#0001 => server waiting for client to establish connection
------------------------------------------------------------*)
VAR_IN_OUT
	xStartSend					: BOOL;
	aReceiveBuffer				: ARRAY [0..MAX_RECEIVE_TCP_SERVER] OF BYTE;
	diReceiveCount				: DINT;
END_VAR

VAR
	m_State    					: BYTE:= 0;
	m_ReceiveBuffer				: ARRAY [0..MAX_RECEIVE_TCP_SERVER_SOCKET] OF BYTE;
	m_ServerSocket				: DINT:= SOCKET_INVALID;
	m_Socket					: DINT:= SOCKET_INVALID;
	m_AddressInfo				: SOCKADDRESS;
	m_BytesReceived				: DINT;
	m_diReturn					: DINT;
	m_xReturn					: BOOL;
	m_SizeSockadr				: DWORD;
	m_ConnectionWatchdog		: TON;
	m_Flags						: DINT;
	m_NoneBlocking   			: DINT:= 1;
	m_Blocking   				: DINT:= 0;
	i							: INT;
	m_count						: DINT;
	diOption					: DINT := 1;
	on: DINT;
END_VAR
IF xEnable THEN
	CASE m_State OF
		STATE_INIT:
			(* Create Socket *)
			m_ServerSocket:= SysSockCreate( SOCKET_AF_INET, SOCKET_STREAM, 0);
			IF m_ServerSocket = SOCKET_INVALID THEN
				(* *)
				diError:= 16#8001;
				m_State:= STATE_ERROR_TRAP;
				RETURN;
			ELSE
				;
			END_IF
			(* Address bindings *)
			(********************)
			on:=1;
			SysSockSetOption( m_ServerSocket, SOCKET_SOL, SOCKET_SO_REUSEADDR, ADR(on), SIZEOF(on) );

			m_AddressInfo.sin_family:= SOCKET_AF_INET;
			m_AddressInfo.sin_port  := SysSockHtons( wPortNumber);
			m_AddressInfo.sin_addr  := SOCKET_INADDR_ANY;
			IF NOT SysSockBind( m_ServerSocket, ADR(m_AddressInfo), SIZEOF(m_AddressInfo)) THEN
				diError:= 16#8002;
				m_State:= STATE_ERROR_TRAP;
				RETURN;
			END_IF
			(* Wait for connections *)
			(************************)
			IF NOT SysSockListen( m_ServerSocket, 1) THEN
				diError:= 16#8003;
				m_State:= STATE_ERROR_TRAP;
			END_IF

			(* Puts SOCKET in NonBlocking mode *)
			m_diReturn:= SysSockIoctl( m_ServerSocket, SOCKET_FIONBIO, ADR(m_NoneBlocking));

			m_State:= STATE_OPEN;


		STATE_OPEN: 	(* Waiting for incomming connection *)
				m_SizeSockadr:=SIZEOF(m_AddressInfo);
				m_Socket:= SysSockAccept( m_ServerSocket, ADR(m_AddressInfo), ADR(m_SizeSockadr));
				diError:=State_open;
				IF m_Socket <> SOCKET_INVALID THEN
					xClientConnected:=TRUE;
					(*Set Push-Bit:new V1.5*)
					IF ADR(%MW0)=16#30000000  OR ADR(%MW0)=16#20000000 THEN (*841 or 881*)
						SysSockSetOption(
							diSocket:=m_Socket,
							diLevel:=6,
							diOption:=SOCKET_TCP_NODELAY,
							pOptionValue:=ADR(diOption),
							diOptionLength:=SIZEOF(diOption));
					ELSE
							;
					END_IF
					SysSockIoctl( m_Socket, SOCKET_FIONBIO, ADR(m_NoneBlocking));
					m_State:= STATE_RX;
					diError:=0;
				END_IF

		STATE_RX:
					m_BytesReceived:= SysSockRecv( m_Socket, ADR(m_ReceiveBuffer), SIZEOF(m_ReceiveBuffer), 0);
					CASE m_BytesReceived OF
					-1:(*no data available or error occured*)
						m_ConnectionWatchdog(IN:=TRUE , PT:=tServerTimeOut );
						IF m_connectionWatchdog.Q THEN
							m_State:= STATE_CLOSE;
							m_ConnectionWatchdog(IN:=FALSE);(*reset connection watchdog*)
							diError := 16#8009;
						END_IF
					0:(* socket was "gracefully closed"  *)
						m_State:= STATE_CLOSE;
						diError := 16#8003;
					ELSE
						(* Copy received data into receive buffer *)
						(********************************)
						FOR i:= 0 TO DINT_TO_INT(m_BytesReceived	)-1 DO
							aReceiveBuffer[diReceiveCount]:= m_ReceiveBuffer[i];
							diReceiveCount:=(diReceiveCount+1) MOD SIZEOF(aReceiveBuffer);
						END_FOR

						m_ConnectionWatchdog(IN:=FALSE);(*reset connection watchdog*)
					END_CASE

				(*send data*)
				IF xStartSend	 THEN
					m_State := STATE_TX;
				END_IF

	STATE_TX:	 (* send TCP-message *)
		m_diReturn := SysSockSend(diSocket := m_Socket,
								  pbyBuffer := ADR(ptSendData^[m_count]),(*geändert V1.4 bisher: [0] *)
								  diBufferSize := diSendCount-m_count,
								  diFlags :=m_Flags);
		CASE m_diReturn OF
		-1:	(* ERROR or data could not yet be send (V1.3 due to new FW11) *)
			m_ConnectionWatchdog(IN:=TRUE , PT:=tServerTimeOut );
			IF m_connectionWatchdog.Q THEN
				m_State:= STATE_CLOSE;
				m_ConnectionWatchdog(IN:=FALSE);(*reset connection watchdog*)
				diError := 16#8007;
			END_IF
		0: (* socket was "gracefully closed"  *)
			m_State := STATE_CLOSE;
			diError := 16#8003;
		ELSE (* succesful *)
			m_count:=m_count+m_diReturn;
			IF m_count>=diSendCount THEN
				diError := 16#0000;
				m_State := STATE_RX;
				m_count:=0;
				xStartSend:=FALSE;
			END_IF
			m_ConnectionWatchdog(IN:=FALSE);(*reset connection watchdog*)
		END_CASE


		STATE_CLOSE:	(* Close the server *)

		IF ADR(%MW0)=16#30000000  OR ADR(%MW0)=16#20000000 THEN (*841 or 881*)
			;
		ELSE
			IF m_Socket>=0 THEN
				SysSockShutdown(m_Socket, 0);;(*870*)
			END_IF
		END_IF
		IF m_Socket>=0 THEN
			SysSockClose( m_Socket);
		END_IF
		xClientConnected:= FALSE;
		m_State:= STATE_OPEN; (* Try to open the server again *)
		m_ConnectionWatchdog(IN:=FALSE);(*reset connection watchdog*)

		STATE_ERROR_TRAP: (* Error Read/Write socket  *)
			m_State:= STATE_ERROR_TRAP;

	ELSE  (* Bad FSM code trap  *)
			m_State:= STATE_ERROR_TRAP;
			diError:= 16#8008;
	END_CASE;
ELSE
	IF m_State <> STATE_INIT THEN
		IF ADR(%MW0)=16#30000000  OR ADR(%MW0)=16#20000000 THEN (*841 or 881*)
			;
		ELSE
			IF m_Socket>=0 THEN
				SysSockShutdown(m_Socket, 0);;(*870*)
			END_IF
		END_IF
		IF m_Socket>=0 THEN
			SysSockClose( m_Socket);
		END_IF
		IF ADR(%MW0)=16#30000000  OR ADR(%MW0)=16#20000000 THEN (*841 or 881*)
			;
		ELSE
			IF m_ServerSocket>=0 THEN
				SysSockShutdown(m_ServerSocket, 0);;(*870*)
			END_IF
		END_IF
		IF m_ServerSocket>=0 THEN
			SysSockClose( m_ServerSocket);
		END_IF
		xClientConnected:= FALSE;
		diError:= 0;
		m_State:= STATE_init; (* Try to open the server again *)
		m_ConnectionWatchdog(IN:=FALSE);(*reset connection watchdog*)
	END_IF
END_IF
END_FUNCTION_BLOCK

(* POU Utils Functions/ADDSTRING, ST *)
FUNCTION ADDSTRING : BOOL
VAR_INPUT
	pTxData: POINTER TO BYTE;
	pString: POINTER TO BYTE;
END_VAR
VAR_IN_OUT
	TxLen: DINT;
END_VAR
VAR
END_VAR
pTxData:=pTxData+TxLen;
WHILE pString^<>0 DO
	pTxData^:=pString^;
	pString:=pString+1;
	pTxData:=pTxData+1;
	TxLen:=TxLen+1;
END_WHILE
END_FUNCTION

(* POU Utils Functions/HEXTORAW, ST *)
FUNCTION HEXTORAW : WORD
VAR_INPUT
	pString		: POINTER TO BYTE;
	StringLen	: WORD;
	pData		: POINTER TO BYTE;
END_VAR
VAR
	xl: WORD;
	xi: WORD;
	xr: BYTE;
END_VAR
xl:=0;
xi:=0;

WHILE xi<StringLen DO

	IF pString^>=97 AND pString^<=102 THEN
		xr := pString^ - 87;
	ELSIF pString^>=65 AND pString^<=70 THEN
		xr := pString^ - 55;
	ELSIF pString^>=48 AND pString^<=57 THEN
		xr := pString^ - 48;
	ELSE
		xr := 16;
	END_IF

	IF xr<16 THEN
		IF (xi AND 1)=0 THEN
			pData^ := xr * 16;
		ELSE
			pData^ := pData^ + xr;
			pData := pData + 1;
			xl := xl + 1;
		END_IF
	END_IF

	xi := xi + 1;
	pString := pString + 1;

END_WHILE

HEXTORAW:=xl;
END_FUNCTION

(* POU Utils/USRLED_Update, ST *)
PROGRAM USRLED_Update
VAR
	OldStatus: en_SYS_Status;

	aFS : ARRAY [0..24] OF FLASHING_SEQUENCE :=
		(Colour:=GREEN,  Frequency:=1,   Relation:=128, Duration:=t#0s,    NextIndex:=0),  (* 0 => RUNNING *)
		(Colour:=ORANGE, Frequency:=1,   Relation:=128, Duration:=t#0s,    NextIndex:=1),  (* 1 => INIT *)
		(Colour:=RED,    Frequency:=4,   Relation:=128, Duration:=t#0s,    NextIndex:=2),  (* 2 => ERROR *)
		(Colour:=RED,    Frequency:=10,  Relation:=128, Duration:=t#0s,    NextIndex:=3),  (* 3 => ALARM *)
		(Colour:=ORANGE, Frequency:=200, Relation:=16,  Duration:=t#100ms, NextIndex:=11), (* 10 *)
		(Colour:=ORANGE, Frequency:=200, Relation:=32,  Duration:=t#100ms, NextIndex:=12),
		(Colour:=ORANGE, Frequency:=200, Relation:=64,  Duration:=t#100ms, NextIndex:=13),
		(Colour:=ORANGE, Frequency:=200, Relation:=128, Duration:=t#100ms, NextIndex:=14),
		(Colour:=ORANGE, Frequency:=200, Relation:=192, Duration:=t#100ms, NextIndex:=15),
		(Colour:=ORANGE, Frequency:=200, Relation:=128, Duration:=t#100ms, NextIndex:=16),
		(Colour:=ORANGE, Frequency:=200, Relation:=64,  Duration:=t#100ms, NextIndex:=17),
		(Colour:=ORANGE, Frequency:=200, Relation:=32,  Duration:=t#100ms, NextIndex:=18),
		(Colour:=ORANGE, Frequency:=200, Relation:=16,  Duration:=t#100ms, NextIndex:=19),
		(Colour:=ORANGE, Frequency:=200, Relation:=8,   Duration:=t#100ms, NextIndex:=10),
		(Colour:=GREEN,  Frequency:=200, Relation:=16,  Duration:=t#100ms, NextIndex:=21), (* 20 *)
		(Colour:=GREEN,  Frequency:=200, Relation:=32,  Duration:=t#100ms, NextIndex:=22),
		(Colour:=GREEN,  Frequency:=200, Relation:=64,  Duration:=t#100ms, NextIndex:=23),
		(Colour:=GREEN,  Frequency:=200, Relation:=128, Duration:=t#100ms, NextIndex:=24),
		(Colour:=GREEN,  Frequency:=200, Relation:=192, Duration:=t#100ms, NextIndex:=25),
		(Colour:=GREEN,  Frequency:=200, Relation:=128, Duration:=t#100ms, NextIndex:=26),
		(Colour:=GREEN,  Frequency:=200, Relation:=64,  Duration:=t#100ms, NextIndex:=27),
		(Colour:=GREEN,  Frequency:=200, Relation:=32,  Duration:=t#100ms, NextIndex:=28),
		(Colour:=GREEN,  Frequency:=200, Relation:=16,  Duration:=t#100ms, NextIndex:=29),
		(Colour:=GREEN,  Frequency:=200, Relation:=8,   Duration:=t#100ms, NextIndex:=20);

	pFS : POINTER TO FLASHING_SEQUENCE;


END_VAR
IF Sys.Status <> OldStatus THEN

	OldStatus:=Sys.Status;

	CASE OldStatus OF

		S_STARTUP:
			pFS:=ADR(aFS);
			SET_FLASHING_SEQUENCE(EN:=TRUE, POINTER_TO_POINTER_TO_ARRAY:=ADR(pFS));
			SET_FLASHING_SEQUENCE_INDEX(EN:=TRUE, IMMEDIATE:=FALSE, INDEX:=1);
			START_FLASHING_SEQUENCE(EN:=TRUE);

		S_RUNNING:
			SET_FLASHING_SEQUENCE_INDEX(EN:=TRUE, IMMEDIATE:=TRUE, INDEX:=0);

	END_CASE

END_IF
END_PROGRAM

(* POU Configuration/MODBUS_CONFIGURATION, ST *)
PROGRAM MODBUS_CONFIGURATION        
VAR                                
END_VAR                            
(*                                 
   <?xml version="1.0" encoding="UTF-16" standalone="yes"?>
<network xml_structure_version="1">
	<generator_settings minRTUTaskCycleTimeMs="5" minEthaskCycleTimeMs="5" ethSlaveMultiplier="0.1" rtuInterfaceMultiplier="0.1" taskGeneration="false"/>
</network>
                              
*)                                 
;                                  
END_PROGRAM

(* POU Plant/SYS_Proc, ST *)
PROGRAM SYS_Proc
VAR
(*	fALARM_PB		:FLT_TAP;
	fALARM_TB		:FLT_TAP;
	fALARM_PM		:FLT_TAP; *)

(*	fGZB_ST			:FLT_TAP;  (* GATEWAY ZIGBEE *)*)
(*	fVPN_ST1		:FLT_TAP;  (* VPN CONNECT *)*)
	fVPN_ST2		:FLT_TAP;  (* VPN STATUS *)
(*	fKEY_CT_ST		:FLT_TAP;  (* DOOR1 *)*)
(*	fKEY_SCT_ST		:FLT_TAP;  (* DOOR2 *)*)
	fKEY_QE_ST		:FLT_TAP;  (* DOOR3 *)

END_VAR
(*************** ISPESL *****************)
(*
fALARM_PB(IN:=ALARM_PB);
IF fALARM_PB.EVH THEN
	LogEv(EL_AlarmStop,EO_PBV,1,1,'Over_Pressure_Alarm');
END_IF

fALARM_TB(IN:=ALARM_TB);
IF fALARM_TB.EVH THEN
	LogEv(EL_AlarmStop,EO_TBV,1,1,'Over_Temperature_Alarm');
END_IF

fALARM_PM(IN:=ALARM_PM);
IF fALARM_PM.EVH THEN
	LogEv(EL_AlarmStop,EO_PMV,1,1,'Under_Pressure_Alarm');
END_IF
*)
(****************************************)

(*### VPN Connection Check ###*)(*
fVPN_ST1(IN:=VPN_ST1);
IF fVPN_ST1.EVH THEN
	LogEv(EL_Log,EO_VPN,1,1,'CONNECT_ON');
END_IF
IF fVPN_ST1.EVL THEN
	LogEv(EL_Log,EO_VPN,1,2,'CONNECT_OFF');
END_IF
*)
(*### VPN Status Check ###*)
fVPN_ST2(IN:=VPN_ST2);
IF fVPN_ST2.EVH THEN
	LogEv(EL_Log,EO_VPN,1,3,'STATUS_UP');
END_IF
IF fVPN_ST2.EVL THEN
	LogEv(EL_Wrn,EO_VPN,1,4,'STATUS_DOWN');
END_IF

(*### DOOR01 Status Check ###*)(*
fKEY_CT_ST(IN:=KEY_CT_ST);
IF fKEY_CT_ST.EVH THEN
	LogEv(EL_Log,EO_DOOR,1,2,'Centrale_termica_Close');
END_IF
IF fKEY_CT_ST.EVL THEN
	LogEv(EL_Wrn,EO_DOOR,1,1,'Centrale_termica_Open');
END_IF
*)
(*### DOOR02 Status Check ###*)(*
fKEY_SCT_ST(IN:=KEY_SCT_ST);
IF fKEY_SCT_ST.EVH THEN
	LogEv(EL_Log,EO_DOOR,2,2,'Sottocentrale_termica_Close');
END_IF
IF fKEY_SCT_ST.EVL THEN
	LogEv(EL_Wrn,EO_DOOR,2,1,'Sottocentrale_termica_Open');
END_IF
*)
(*### DOOR03 Status Check ###*)
fKEY_QE_ST(IN:=KEY_QE_ST);
IF fKEY_QE_ST.EVH THEN
	LogEv(EL_Log,EO_DOOR,3,2,'Quadro_Close');
END_IF
IF fKEY_QE_ST.EVL THEN
	LogEv(EL_Wrn,EO_DOOR,3,1,'Quadro_Open');
END_IF
END_PROGRAM

(* POU Utils Functions/FLT_TAP, ST *)
FUNCTION_BLOCK FLT_TAP
VAR_INPUT
	IN		: BOOL;
	TAP		: BYTE:=4;
	INITEV	: BOOL:=TRUE;
END_VAR
VAR_OUTPUT
	OUT		: BOOL;
	EVH		: BOOL;
	EVL		: BOOL;
END_VAR
VAR
	init	: BOOL:=FALSE;
	cnt		: BYTE;
END_VAR
EVH:=FALSE;
EVL:=FALSE;

IF NOT init THEN
	init := TRUE;
	IF INITEV THEN
		OUT  := NOT IN;
		cnt  := TAP;
	ELSE
		OUT  := IN;
	END_IF
END_IF

IF OUT<>IN THEN
	cnt:=cnt+1;
	IF cnt>TAP THEN
		OUT:=IN;
		cnt:=0;
		IF OUT THEN EVH:=TRUE; ELSE EVL:=TRUE; END_IF
	END_IF
ELSE
	cnt:=0;
END_IF
END_FUNCTION_BLOCK

(* POU TCP_Logger/LogEv, ST *)
FUNCTION LogEv : BOOL
VAR_INPUT
	Level	: en_Logger_ErrLev;
	Object  : en_SYS_Objects;
	Index	: WORD;
	Error	: WORD;
	Message : STRING;
END_VAR
VAR
	s1 : STRING(160);
	i  : INT;
END_VAR
(* Execute error level operations *)
CASE Level OF
	EL_Wrn: 		Sys.Warning:=TRUE;
	EL_Alarm: 		Sys.Alarm:=TRUE;
	EL_AlarmStop: 	Sys.Alarm:=TRUE; (* GO TO STOP STATE!! *)
END_CASE

(* Fill lastlog list *)
s1:=CONCAT(Sys.Time_LogString,';Lev=');
s1:=CONCAT(s1,INT_TO_STRING(Level));
s1:=CONCAT(s1,';Obj=');
s1:=CONCAT(s1,INT_TO_STRING(Object));
s1:=CONCAT(s1,';Idx=');
s1:=CONCAT(s1,WORD_TO_STRING(Index));
s1:=CONCAT(s1,';Err=');
s1:=CONCAT(s1,WORD_TO_STRING(Error));
Sys.LastLogs_Dat[Sys.LastLogs_Idx]:=s1;
Sys.LastLogs_Msg[Sys.LastLogs_Idx]:=Message;
Sys.LastLogs_Idx:=Sys.LastLogs_Idx+1;
IF Sys.LastLogs_Idx>5 THEN Sys.LastLogs_Idx:=0; END_IF

(*---------------------------------------------------------------*)
(*---------------------------------------------------------------*)
Logger.TLen:=0;
(* Set GET header *)
ADDSTRING(ADR(Logger.TData), ADR(Logger_GETSTART), Logger.TLen);

(* Insert Header *)
s1:=INSERT('ID=&V=1&D=',DWORD_TO_STRING(Plant_SN),3);
s1:=CONCAT(s1,Sys.Time_LogString);
s1:=CONCAT(s1,'&S=');
IF Sys.Alarm THEN i:=2; ELSIF Sys.Warning THEN i:=1; ELSE i:=0; END_IF
s1:=CONCAT(s1,INT_TO_STRING(i));
ADDSTRING(ADR(Logger.TData), ADR(s1), Logger.TLen);

(* Insert ERR *)
s1:=CONCAT('&ERR=',INT_TO_STRING(Level));
s1:=CONCAT(s1,';');
s1:=CONCAT(s1,INT_TO_STRING(Object));
s1:=CONCAT(s1,';');
s1:=CONCAT(s1,WORD_TO_STRING(Index));
s1:=CONCAT(s1,';');
s1:=CONCAT(s1,WORD_TO_STRING(Error));
s1:=CONCAT(s1,';');
ADDSTRING(ADR(Logger.TData), ADR(s1), Logger.TLen);
s1:=Message;
ADDSTRING(ADR(Logger.TData), ADR(s1), Logger.TLen);

(* Finalize string *)
ADDSTRING(ADR(Logger.TData), ADR(Logger_GETEND), Logger.TLen);

(*---------------------------------------------------------------*)
(*---------------------------------------------------------------*)

Logger_Send();
END_FUNCTION

(* POU TCP_Logger/Logger_Send, ST *)
FUNCTION Logger_Send : BOOL
VAR
	hFile: 	DWORD;
	pos:	DWORD;
END_VAR
(* Read log position *)
pos:=SysFileGetSize(Logger_DataFile);
(* Check log size, bckup and erase if no pending messages *)
IF pos>100000000 (*100M*) THEN
	hFile:=SysFileOpen(Logger_IndexFile,'r');
	IF hFile=0 THEN
		SysFileDelete(Logger_DataFileOld);
		SysFileRename(Logger_DataFile,Logger_DataFileOld);
		pos:=0;
	ELSE
		SysFileClose(hFile);
	END_IF
END_IF
(* Write message on log file *)
hFile:=SysFileOpen(Logger_DataFile,'a');
IF hFile<>0 THEN
	SysFileWrite(hFile, ADR(Logger.TData), Logger.TLen);
	SysFileClose(hFile);
ELSE
	Sys.Warning:=TRUE;
END_IF


(* Check logger status *)
IF Logger.SendReq=FALSE THEN
	(* Set log position for recovery *)
	Logger.SendIdx:=pos;
	(* Copy message data *)
	MEMCPY(ADR(Logger.TData),ADR(Logger.SendData),DINT_TO_WORD(Logger.TLen));
	Logger.SendLen:=Logger.TLen;
	(* Trigger request *)
	Logger.SendReq:=TRUE;
ELSE
	(* Add message position+size in recovery indexes *)
	hFile:=SysFileOpen(Logger_IndexFile,'a');
	SysFileWrite(hFile, ADR(pos), SIZEOF(pos));
	SysFileWrite(hFile, ADR(Logger.TLen), SIZEOF(Logger.TLen));
	SysFileClose(hFile);
END_IF
END_FUNCTION

(* POU Utils Functions/MEMCPY, ST *)
FUNCTION MEMCPY:BOOL
VAR_INPUT
	pSourceAddress:POINTER TO ARRAY[1..2] OF BYTE;
	pDestinationAddress:POINTER TO ARRAY[1..2] OF BYTE;
	BytesToCopy:WORD;
END_VAR
VAR
END_VAR
WHILE (BytesToCopy > 0) DO
	pDestinationAddress^[1]:=pSourceAddress^[1]; (* copy bytes from source to destination *)
	pDestinationAddress:=ADR(pDestinationAddress^[2]); (* increment destination *)
	pSourceAddress:=ADR(pSourceAddress^[2]);(* increment source *)
	BytesToCopy:=BytesToCopy -1; (* decrement number of bytes to copy *)
END_WHILE
END_FUNCTION

(* POU Utils Functions/AVERAGE_T, ST *)
FUNCTION_BLOCK AVERAGE_T
VAR_INPUT
	IN: 	INT;
END_VAR
VAR_OUTPUT
	HI:		INT;
	AVG:	INT;
	LOW:	INT;
	ERR:	BOOL;
END_VAR
VAR
	sum:	DINT;
	cnt:	WORD;
END_VAR
IF cnt>=65000 THEN
	ERR:=TRUE;
	Read();
	sum := sum - AVG;
	cnt := cnt + 1;
END_IF

sum := sum + IN;
cnt := cnt + 1;

IF IN<LOW THEN  LOW:=IN; END_IF
IF IN>HI  THEN HI :=IN; END_IF
END_FUNCTION_BLOCK
ACTION Read:
AVG := DINT_TO_INT(sum/cnt);
END_ACTION
ACTION Reset:
HI:=IN;
AVG:=IN;
LOW:=IN;
ERR:=FALSE;

sum:=IN;
cnt:=1;
END_ACTION

(* POU Utils/CSV_Log, ST *)
FUNCTION CSV_Log : BOOL
VAR_INPUT
END_VAR
VAR CONSTANT
	LogFileName:STRING:='S:\LOGS_ID3V3.CSV';
END_VAR
VAR
	s1 : STRING(180);
	hFile: 	DWORD;
END_VAR
(* Check file presence *)
hFile:=SysFileOpen(LogFileName,'r');
IF hFile=0 THEN
	(*** File not exist *** Create file and write header *)
	hFile:=SysFileOpen(LogFileName,'w');
	IF hFile<>0 THEN
		(* Write CSV header *)
		s1:='DATE-TIME;T-SA;T-S02;T-S03;T-S04;T-S05;T-S06;T-S07;';
		SysFileWrite(hFile, ADR(s1), LEN(s1));
		s1:='PORT01-Flow;PORT01-Cnt;GAS01-Cnt;GAS02-Cnt;';
		SysFileWrite(hFile, ADR(s1), LEN(s1));
		s1:='CTB250-Power;CTB250-KWH;CTB250-GWH';
		SysFileWrite(hFile, ADR(s1), LEN(s1));
		SysFileWrite(hFile, ADR(Logger_CRLF), LEN(Logger_CRLF));
	END_IF
ELSE
	(*** File exist *** Close file and reopen in append mode *)
	SysFileClose(hFile);
	hFile:=SysFileOpen(LogFileName,'a');
END_IF

(* Log to file *)
IF hFile<>0 THEN
	(* Date stamp *)
	s1:=REPLACE( Sys.Time_LogString , ' ' , 1 , 11 );
	SysFileWrite(hFile, ADR(s1), LEN(s1));
	(* Log data *)
	s1:=CONCAT(';', INT_TO_STRING(TT_S01) );
	s1:=CONCAT(s1 , ';' );
	s1:=CONCAT(s1 , INT_TO_STRING(TPV02.ValoreScalato) );
	s1:=CONCAT(s1 , ';' );
	s1:=CONCAT(s1 , INT_TO_STRING(TPV03.ValoreScalato) );
	s1:=CONCAT(s1 , ';' );
	s1:=CONCAT(s1 , INT_TO_STRING(TPV04.ValoreScalato) );
	s1:=CONCAT(s1 , ';' );
	s1:=CONCAT(s1 , INT_TO_STRING(TPV05.ValoreScalato) );
	s1:=CONCAT(s1 , ';' );
	s1:=CONCAT(s1 , INT_TO_STRING(TPV06.ValoreScalato) );
	s1:=CONCAT(s1 , ';' );
	s1:=CONCAT(s1 , INT_TO_STRING(TPV07.ValoreScalato) );
	SysFileWrite(hFile, ADR(s1), LEN(s1));
	s1:=CONCAT(';', INT_TO_STRING(PORT01.ValoreScalato) );
	s1:=CONCAT(s1 , ';' );
	s1:=CONCAT(s1 , DINT_TO_STRING(PortataTotalePORT01) );
	s1:=CONCAT(s1 , ';' );
	s1:=CONCAT(s1 , DINT_TO_STRING(PortataTotaleGAS01) );
	s1:=CONCAT(s1 , ';' );
	s1:=CONCAT(s1 , DINT_TO_STRING(PortataTotaleGAS02) );
	SysFileWrite(hFile, ADR(s1), LEN(s1));
	s1:=CONCAT(';', DINT_TO_STRING(REAL_TO_DINT(CTB250.POWER_KW)) );
	s1:=CONCAT(s1 , ';' );
	s1:=CONCAT(s1 , DWORD_TO_STRING(CTB250_ENERGY) );
	SysFileWrite(hFile, ADR(s1), LEN(s1));

	(* Add line CRLF and close *)
	SysFileWrite(hFile, ADR(Logger_CRLF), LEN(Logger_CRLF));
	SysFileClose(hFile);
END_IF
END_FUNCTION

(* POU Utils Functions/FLT_EVENT, ST *)
FUNCTION_BLOCK FLT_EVENT
VAR_INPUT
	IN		: BOOL;
	INITEV	: BOOL:=TRUE;
END_VAR
VAR_OUTPUT
	EVH		: BOOL;
	EVL		: BOOL;
END_VAR
VAR
	init	: BOOL:=FALSE;
	old		: BOOL;
END_VAR
EVH:=FALSE;
EVL:=FALSE;

IF NOT init THEN
	init:=TRUE;
	IF INITEV THEN
		old := NOT IN;
	ELSE
		old := IN;
	END_IF
END_IF

IF old<>IN THEN
	old:=IN;
	IF IN THEN EVH:=TRUE; ELSE EVL:=TRUE; END_IF
END_IF
END_FUNCTION_BLOCK

(* POU Utils Functions/LINEAR, ST *)
FUNCTION LINEAR : INT (* Linear interpolation *)
VAR_INPUT
	PuntoMinX:INT;
	PuntoMaxX:INT;
	ValIn : INT;
	PuntoMinY:REAL;
	PuntoMaxY:REAL;
	Decimali: BYTE;
END_VAR
VAR
	Gain: REAL;
	PuntoMinX_R	:REAL;
	PuntoMaxX_R	:REAL;
	Linearizzazione_R:REAL;
END_VAR
PuntoMinX_R:=INT_TO_REAL(PuntoMinX);
PuntoMaxX_R:=INT_TO_REAL(PuntoMaxX);

Gain:=(PuntoMaxX_R-PuntoMinX_R)/(PuntoMaxY-PuntoMinY);	(* Calcolo in guadagno per la linarizzazione *)
Linearizzazione_R:=PuntoMinx+(Gain*(ValIn-PuntoMinY));	(* Ottengo il valore linearizzato *)

LINEAR:=REAL_TO_INT(Linearizzazione_R*(EXPT(10, Decimali)));  (* Ottengo intero con i decimai voluti *)
END_FUNCTION

(* POU TCP_Logger/LogTrig, ST *)
FUNCTION LogTrig : BOOL
VAR
	s1 : STRING(160);
	i  : BYTE;
END_VAR
(*---------------------------------------------------------------*)
(*---------------------------------------------------------------*)
Logger.TLen:=0;
(* Set GET header *)
ADDSTRING(ADR(Logger.TData), ADR(Logger_GETSTART), Logger.TLen);

(* Insert Header *)
s1:=INSERT('ID=&V=1&D=',DWORD_TO_STRING(Plant_SN),3);
s1:=CONCAT(s1,Sys.Time_LogString);
s1:=CONCAT(s1,'&S=');
IF Sys.Alarm THEN i:=2; ELSIF Sys.Warning THEN i:=1; ELSE i:=0; END_IF
s1:=CONCAT(s1,BYTE_TO_STRING(i));
ADDSTRING(ADR(Logger.TData), ADR(s1), Logger.TLen);

(* Insert TPVs *)
s1:=CONCAT('&TPV=',INT_TO_STRING(TPV01.IN));
s1:=CONCAT(s1,';'); s1:=CONCAT(s1,INT_TO_STRING(TPV02.ValoreScalato));
s1:=CONCAT(s1,';'); s1:=CONCAT(s1,INT_TO_STRING(TPV03.ValoreScalato));
s1:=CONCAT(s1,';'); s1:=CONCAT(s1,INT_TO_STRING(TPV04.ValoreScalato));
s1:=CONCAT(s1,';'); s1:=CONCAT(s1,INT_TO_STRING(TPV05.ValoreScalato));
s1:=CONCAT(s1,';'); s1:=CONCAT(s1,INT_TO_STRING(TPV06.ValoreScalato));
s1:=CONCAT(s1,';'); s1:=CONCAT(s1,INT_TO_STRING(TPV07.ValoreScalato));
ADDSTRING(ADR(Logger.TData), ADR(s1), Logger.TLen);

(* Insert contabilizers  *)
s1:=CONCAT('&PORT01=',INT_TO_STRING(PORT01.ValoreScalato));
s1:=CONCAT(s1,';'); s1:=CONCAT(s1,DINT_TO_STRING(PortataTotalePORT01));
s1:=CONCAT(s1,';'); s1:=CONCAT(s1,BYTE_TO_STRING(PORT01.Status_Log));
ADDSTRING(ADR(Logger.TData), ADR(s1), Logger.TLen);

s1:=CONCAT('&GAS01=',DINT_TO_STRING(PortataTotaleGAS01));
s1:=CONCAT(s1,';'); s1:=CONCAT(s1,BYTE_TO_STRING(GAS01.Status_Log));
ADDSTRING(ADR(Logger.TData), ADR(s1), Logger.TLen);

s1:=CONCAT('&GAS02=',DINT_TO_STRING(PortataTotaleGAS02));
s1:=CONCAT(s1,';'); s1:=CONCAT(s1,BYTE_TO_STRING(GAS02.Status_Log));
ADDSTRING(ADR(Logger.TData), ADR(s1), Logger.TLen);

(* Insert active contabilizers *)
FOR i := 0 TO CTBSCAN01.EndScanAddress  DO
	IF 	CTBSCAN01.NodoMBusPresente[i]=TRUE THEN
		s1:=INSERT('&CTB=',BYTE_TO_STRING(i),4);
		s1:=CONCAT(s1,';'); s1:=CONCAT(s1,'0' (*CTBSCAN01.CTB_utFTemp [i].Value*) );
		s1:=CONCAT(s1,';'); s1:=CONCAT(s1,'0' (*CTBSCAN01.CTB_utRTemp [i].Value*) );
		s1:=CONCAT(s1,';'); s1:=CONCAT(s1,'0' (*CTBSCAN01.CTB_utFlow  [i].Value*) );
		s1:=CONCAT(s1,';'); s1:=CONCAT(s1,'0' (*CTBSCAN01.CTB_utPower [i].Value*) );
		s1:=CONCAT(s1,';'); s1:=CONCAT(s1,'0' (*CTBSCAN01.CTB_utEnergy[i].Value*) );
		s1:=CONCAT(s1,';'); s1:=CONCAT(s1,BYTE_TO_STRING(CTBSCAN01.Status_Log_NodoMBus[i]));
		ADDSTRING(ADR(Logger.TData), ADR(s1), Logger.TLen);
	END_IF
END_FOR

(* Insert static contabilizers *)
s1:=INSERT('&CTB=',BYTE_TO_STRING(CTB250.ID),4);
					s1:=CONCAT(s1,INT_TO_STRING(CTB250.T_SEND) );
s1:=CONCAT(s1,';'); s1:=CONCAT(s1,INT_TO_STRING(CTB250.T_RET) );
s1:=CONCAT(s1,';'); s1:=CONCAT(s1,DWORD_TO_STRING(INT_TO_DWORD(CTB250.FLOW)*1000) );
s1:=CONCAT(s1,';'); s1:=CONCAT(s1,DWORD_TO_STRING(REAL_TO_DWORD(CTB250.POWER_KW*1000)) );
s1:=CONCAT(s1,';'); s1:=CONCAT(s1,DWORD_TO_STRING(CTB250_ENERGY) );
s1:=CONCAT(s1,';'); s1:=CONCAT(s1,BYTE_TO_STRING(CTB250.Status_Log));
ADDSTRING(ADR(Logger.TData), ADR(s1), Logger.TLen);

(* Finalize string *)
ADDSTRING(ADR(Logger.TData), ADR(Logger_GETEND), Logger.TLen);

(*---------------------------------------------------------------*)
(*---------------------------------------------------------------*)

Logger_Send();
END_FUNCTION

(* POU Utils Functions/MEMCLR, ST *)
FUNCTION MEMCLR:BOOL
VAR_INPUT
	pDestinationAddress:POINTER TO ARRAY[1..2] OF BYTE;
	BytesToClear:WORD;
END_VAR
VAR
END_VAR
WHILE (BytesToClear > 0) DO
	pDestinationAddress^[1]:=0;
	pDestinationAddress:=ADR(pDestinationAddress^[2]); (* increment destination *)
	BytesToClear:=BytesToClear -1; (* decrement number of bytes to copy *)
END_WHILE
END_FUNCTION

(* POU Plant_Objects/obj_GAS, ST *)
FUNCTION_BLOCK obj_GAS
VAR_INPUT
	(* Settings *)
	ID				: BYTE;
	DI_Input		: BOOL;	(* Ingresso Digitale per il conteggio  *)
	Peso			: INT;	(* Peso dell' impulso , serve per avere una lettura immediata dell'unità ingegneristica *)
	TempoTimeOut	: TIME;	(* Minuti di inattività per la segnalazione del WRN *)
END_VAR
VAR_OUTPUT
	WRN				: BOOL;	(* Segnalazione Warning *)
	(* Status *)
	Status_Log		: BYTE;
	Status_Vis 		: DWORD;
END_VAR
VAR
	TRig_DI			: R_TRIG;
	TimeOut			: TON;
	TRigR_TimeOut	: R_TRIG;
	TRigL_TimeOut	: F_TRIG;
END_VAR
VAR_IN_OUT
                Contatore                          : DINT;
                Totalizzatore    			 :DINT; (* Totale Conteggio x valore peso *)
END_VAR
(* MANCA UN MINIMO DI TAP ==> meglio usare FLT_TAP per detect fronte di salita *)

(* Triggero sul fronte di salita l'ingresso digitale *)
TRig_DI(CLK:=DI_Input );

(* Conto i fronti di salita  in modo de creare rapporto*)
IF  TRig_DI.Q THEN
	Contatore:=Contatore+1;
	Totalizzatore:=Contatore*Peso;
END_IF

(* Imposto il time out se non c'è movimento sulla linea per il tempo impostato loggo un Warning *)
TimeOut(IN:=NOT DI_Input , PT:=TempoTimeOut, Q=> , ET=> );
TRigR_TimeOut( CLK:= TimeOut.Q  );
TRigL_TimeOut( CLK:= TimeOut.Q  );

		IF  TRigR_TimeOut.Q THEN     (* Condizione di WARNING *)
					WRN:=TRUE;
					Status_Log:=1; Status_Vis:=16#20F0F0;
 					LogEv(EL_Wrn,EO_GAS,ID,2,'Nessun_Movimento');
		END_IF

		IF  TRigL_TimeOut.Q THEN     (* Condizione di Rientro dal WARNING *)
					WRN:=FALSE;
					Status_Log:=0; Status_Vis:=16#20F020;
 					LogEv(EL_Log,EO_GAS,ID,1,'');
		END_IF
END_FUNCTION_BLOCK

(* POU Plant_Objects/obj_MBUS, ST *)
FUNCTION_BLOCK obj_MBUS
VAR_INPUT
	ID				: BYTE;
	COM				: BYTE;
	BAUDRATE		: COM_BAUDRATE;
	(* Interface *)
	MBus 			: typMBus;
	MBus_Master 	: FbMBusMaster;
END_VAR
VAR_OUTPUT
	(* Status *)
	Status_Log		: BYTE;
	Status_Vis 		: DWORD;
END_VAR
VAR
END_VAR
MBus_Master( bCOMPORT:=COM , enumBAUDRATE:=BAUDRATE , utMBus:=MBus );

(* Check status *)
IF MBus.bCOM_ERROR<>0 THEN Status_Log:=2; Status_Vis:=16#2020F0;
					  ELSE Status_Log:=0; Status_Vis:=16#20F020;
END_IF
END_FUNCTION_BLOCK

(* POU Plant_Objects/obj_MBUS_CTB, ST *)
FUNCTION_BLOCK obj_MBUS_CTB
VAR_INPUT
	ID				: BYTE;
	ADDRESS			: BYTE;
	UpdateNow		: BOOL;
	M1_Start		: BOOL;
END_VAR
VAR_IN_OUT
	MBus			: typMBus;
END_VAR
VAR_OUTPUT
	(* Visu/Log *)
	Status_Log		: BYTE;
	Status_Vis : DWORD;
END_VAR
VAR
	T1				: TON := ( PT:=T#120s );
	M1				: FbMBus_Heat;
	C1				: FbUnitConverter;
END_VAR
(* Auto refresh timer *)
T1( IN:=NOT ( T1.Q OR M1_Start ) );
(* Trigger refresh *)
IF NOT M1_Start AND (T1.Q OR UpdateNow) THEN
	M1_Start:=TRUE;
	UpdateNow:=FALSE;
END_IF

M1(
	dwAdr:=ADDRESS,
	xSND_NKE:=TRUE ,
	utMBus:=MBus ,
	xStart:=M1_Start ,
);


(* Check status *)
IF M1.bError<>0 THEN Status_Log:=2; Status_Vis:=16#2020F0;
			    ELSE Status_Log:=0; Status_Vis:=16#20F020;
END_IF
END_FUNCTION_BLOCK

(* POU Plant_Objects/obj_MBUS_CTB_SCANNER, ST *)
FUNCTION_BLOCK obj_MBUS_CTB_SCANNER
VAR_INPUT
	(* Settings *)
	ID				: BYTE;
	EndScanAddress	: BYTE:=250;
	EndlessRescan   : BOOL:=FALSE;
	ScanPause		: TIME:=t#500ms;
	(* Controls *)
	Refresh			: BOOL; (* Enable automatic refresh of detected CTBs *)
	Rescan			: BOOL; (* Perform complete search for list-update *)
END_VAR
VAR_IN_OUT
	MBUS			: obj_MBUS;
END_VAR
VAR_OUTPUT
	ConnectedCTBs	: BYTE; (* Number of connected CTBs at last rescan *)
	(* Status *)
	Status_Log		: BYTE;
	Status_Vis 		: DWORD;
END_VAR
VAR

	(* Virtual contabilizer for scanner *)
	M1			: FbMBus_Heat;
	M1_Start	: BOOL;

	(* Da definire come datatype *)
(*	CTBS	: ARRAY [0..255] OF typ_MBUS_CTBS; *)
	NodoMBusPresente		: ARRAY [0..255] OF BOOL;
	ErroreNodoMBus			: ARRAY [0..255] OF BYTE;
	Status_Log_NodoMBus		: ARRAY [0..255] OF BYTE;
	Status_Vis_NodoMBus		: ARRAY [0..255] OF DWORD;
	CTB_utMBInfo			: ARRAY [0..255] OF typMBusInfo;
	CTB_utFTemp	 			: ARRAY [0..255] OF typMBusRecord;
	CTB_utRTemp	 			: ARRAY [0..255] OF typMBusRecord;
	CTB_utPower	 			: ARRAY [0..255] OF typMBusRecord;
	CTB_utFlow	 			: ARRAY [0..255] OF typMBusRecord;
	CTB_utEnergy 			: ARRAY [0..255] OF typMBusRecord;
	CTB_utVolume 			: ARRAY [0..255] OF typMBusRecord;
	CTB_utDTemp	 			: ARRAY [0..255] OF typMBusRecord;
	VisuDatiMbus			: ARRAY [0..255] OF typ_VisuStrutturaMbus;

	sta		 : BYTE; 	(* Status: 0:Idle, 1:Wait scan response, 2:Wait refresh response, 3:Wait refresh delay *)
	cnt		 : BYTE;	(* Selection counter *)
	pass_cnt : BYTE;	(* Active counter *)
	dly 	 : TON;
	s1 		 : STRING;
END_VAR
CASE sta OF
	0:
		IF NOT M1_Start THEN
			IF Rescan THEN
				(* Start scanning - with fast timeout and only one retry *)
				cnt:=0;
				pass_cnt:=0;
				MBUS.MBus_Master.bRetries:=1;
				MBUS.MBus_Master.tTimeout:=T#500ms;
				M1.dwAdr:=cnt;
				M1_Start:=TRUE;
				sta:=1;
			ELSIF Refresh THEN
				(* Start refresh *)
				cnt:=0;
				GoToNextActive();
				IF cnt>EndScanAddress THEN
					Refresh:=FALSE;
				ELSE
					MBUS.MBus_Master.bRetries:=3;
					MBUS.MBus_Master.tTimeout:=T#1000ms;
					M1.dwAdr:=cnt;
					M1_Start:=TRUE;
					sta:=2;
				END_IF
			END_IF
		END_IF

	1:
		IF NOT Rescan THEN
			sta:=0;
		ELSE
			IF NOT M1_Start THEN
				(* Get scan result *)
				UpdateNode();
				UpdateVisu();
				(* Next object *)
				cnt:=cnt+1;
				IF cnt>EndScanAddress THEN
					ConnectedCTBs:=pass_cnt;
					Rescan:=EndlessRescan;
					sta:=0;
				ELSE
					M1.dwAdr:=cnt;
					M1_Start:=TRUE;
				END_IF;
			END_IF
		END_IF

	2:
		IF NOT Refresh OR Rescan THEN
			sta:=0;
		ELSE
			IF NOT M1_Start THEN
				(* Get scan result *)
				UpdateNode();
				UpdateVisu();
				(* Next object *)
				cnt:=cnt+1;
				GoToNextActive();
				IF cnt>EndScanAddress THEN
					sta:=3;
					dly(IN:=FALSE, PT:=ScanPause);
				ELSE
					M1.dwAdr:=cnt;
					M1_Start:=TRUE;
				END_IF;
			END_IF
		END_IF

	3:
		(* Refresh cycle delay *)
		dly(IN:=TRUE, PT:=ScanPause);
		IF dly.Q THEN sta:=0; END_IF

ELSE
	sta:=0;
END_CASE

(* Update virtual contabilizer *)
M1( (*dwAdr:= cnt,*) xSND_NKE:=TRUE , utMBus:=MBUS.MBus , xStart:=M1_Start );
END_FUNCTION_BLOCK
ACTION GoToNextActive:
WHILE NodoMBusPresente[cnt] <> TRUE AND cnt<=EndScanAddress DO
	cnt:=cnt+1;
END_WHILE
END_ACTION
ACTION UpdateNode:
ErroreNodoMBus[cnt]:=M1.bError;
CTB_utMBInfo[cnt]:=M1.utMBInfo;
CTB_utEnergy[cnt]:=M1.utEnergy;
CTB_utPower [cnt]:=M1.utPower;
CTB_utVolume[cnt]:=M1.utVolume;
CTB_utFlow  [cnt]:=M1.utFlow;
CTB_utFTemp [cnt]:=M1.utFTemp;
CTB_utRTemp [cnt]:=M1.utRTemp;
CTB_utDTemp [cnt]:=M1.utDTemp;

				(* Check node status *)
				IF ErroreNodoMBus[cnt]<>0  THEN
           			(* se non sono in allarme di comunicazione loggo l'allarme *)
					IF Status_Log_NodoMBus[cnt]<>2 AND sta=2 THEN
						LogEv(EL_Alarm,EO_CTB,cnt,2,CONCAT('Err',BYTE_TO_STRING(ErroreNodoMBus[cnt])));
					END_IF
					(*se sono in fase di rescan memorizzo l'assenza del nodo *)
					IF sta=1 THEN NodoMBusPresente[cnt]:=FALSE;	END_IF
					(* Update status *)
					Status_Log_NodoMBus[cnt]:=2;
					Status_Vis_NodoMBus[cnt]:=16#2020F0;
		    	ELSE
					(* tutto OK Comunizaione andata a buon termine *)
					(* se non sono in allarme di comunicazione loggo l'allarme, ma  se non presente *)
					IF Status_Log_NodoMBus[cnt]<>0 AND sta=2 THEN
						LogEv(EL_Log,EO_CTB,cnt,1,'Nodo_OK');
					END_IF
					(*se sono in fase di rescan memorizzo la presenza del nodo *)
					IF sta=1 THEN NodoMBusPresente[cnt]:=TRUE; pass_cnt:=pass_cnt+1; END_IF
					(* Update status *)
					Status_Log_NodoMBus[cnt]:=0;
					Status_Vis_NodoMBus[cnt]:=16#20F020;
				END_IF
END_ACTION
ACTION UpdateVisu:
VisuDatiMbus[cnt].sdNodoPresente	:=SEL(NodoMBusPresente[cnt],'FAIL!','OK');
VisuDatiMbus[cnt].sdEnergia			:=CTB_utMBInfo[cnt].stMAN;
VisuDatiMbus[cnt].sdPotenza			:=CTB_utMBInfo[cnt].stMED;
VisuDatiMbus[cnt].sdVolume			:=CTB_utMBInfo[cnt].stID;

(*
VisuDatiMbus[cnt].sdEnergia			:=CONCAT(CTB_utEnergy[cnt].Value,CTB_utEnergy[cnt].Unit);
VisuDatiMbus[cnt].sdPotenza			:=CONCAT(CTB_utPower [cnt].Value,CTB_utPower [cnt].Unit);
VisuDatiMbus[cnt].sdVolume			:=CONCAT(CTB_utVolume[cnt].Value,CTB_utVolume[cnt].Unit);
VisuDatiMbus[cnt].sdFlow			:=CONCAT(CTB_utFlow  [cnt].Value,CTB_utFlow  [cnt].Unit);
VisuDatiMbus[cnt].sdTempIngresso	:=CONCAT(CTB_utFTemp [cnt].Value,CTB_utFTemp [cnt].Unit);
VisuDatiMbus[cnt].sdTempaUscita		:=CONCAT(CTB_utRTemp [cnt].Value,CTB_utRTemp [cnt].Unit);
VisuDatiMbus[cnt].sdTempDelta		:=CONCAT(CTB_utDTemp [cnt].Value,CTB_utDTemp [cnt].Unit);
*)

IF sta=1 AND NodoMBusPresente[cnt] THEN
(*	s1:=SEL(NodoMBusPresente[cnt],'FAIL','OK');*)
	s1:='FOUND';
	s1:=CONCAT(s1,'_');
	s1:=CONCAT(s1,CTB_utMBInfo[cnt].stMED);
	s1:=CONCAT(s1,'_');
	s1:=CONCAT(s1,CTB_utMBInfo[cnt].stID);
	LogEv(EL_Log,EO_CTB,cnt,100,s1);
END_IF
END_ACTION

(* POU Plant_Objects/obj_PORT, ST *)
FUNCTION_BLOCK obj_PORT
VAR_INPUT
	(* Settings *)
	ID			: BYTE;
	Peso		 : INT;		(* Peso dell' impulso , serve per avere una lettura immediata dell'unità ingegneristica *)
	TempoTimeOut : TIME;	(* Minuti di inattività per la segnalazione del WRN *)
	PuntoMinX	: INT;  (*Parametri per la scalatura *)
	PuntoMaxX	: INT;
	PuntoMinY	: REAL;
	PuntoMaxY	: REAL;
	Decimali	: BYTE;
	TAP			: INT:=2000;   (* Filtro in msec *)
	INITEV		: BOOL:= TRUE; (* Generate init OK event *)
	SogliaHH	: WORD;    (* Soglia per segnalazione Allarme Extra Range in alto - Solitamente sondo in CC *)
	SogliaHL	: WORD;    (* Soglia per segnalazione Allarme Extra Range in Basso - Solitamente sondo Aperta *)
	SogliaWH	: REAL;    (* Soglia per segnalazione Warning  in alto  *)
	SogliaWL	: REAL;    (* Soglia per segnalazione Warning in basso  *)

	(* Physical inputs *)
	DI_INPUT	: BOOL; (* Ingresso Digitale per il conteggio  *)
	AI_INPUT	: WORD; (* Ingresso Analogico *)
END_VAR
VAR_IN_OUT
    Contatore		: DINT;
    Totalizzatore	: DINT; (* Totale Conteggio x valore peso *)
END_VAR
VAR_OUTPUT
	ValoreScalato	: INT;	(*Valore istantaneo scalato ingresso Analgico *)
	ERR				: BOOL;	(* Segnalazione Errore *)
	WRN				: BOOL;	(* Segnalazione Warning *)

	(* Status *)
	Status_Log	: BYTE;
	Status_Vis 	: DWORD;

END_VAR
VAR
	TRig_DI		: R_TRIG;

	TimeOut		: TON;
	TRigR_TimeOut: R_TRIG;
	TRigL_TimeOut: F_TRIG;

	SegnaleHH: BOOL;
	SegnaleHL: BOOL;
	SegnaleOK: BOOL;

	SegnaleWH: BOOL;
	SegnaleWL: BOOL;

	FiltroWRN:TON;
	FiltroOK:TON;
	FiltroERR:TON;
END_VAR
(**** Gestione ingresso digitale per la contabilizzazzione degli impulsi *****************)

(* TRiggero sul fronte di salita l'ingresso Digitale *)

TRig_DI(CLK:=DI_Input );

(* Conto i fronti di salita  in modo de creare rapporto*)
IF  TRig_DI.Q THEN
	Contatore:=Contatore+1;
	Totalizzatore:=Contatore*Peso;
END_IF


(* Imposto il time out se non c'è movimento sulla linea per il tempo impostato loggo un Warning *)

TimeOut(IN:=NOT DI_Input , PT:=TempoTimeOut, Q=> , ET=> );
TRigR_TimeOut(CLK:= TimeOut.Q  );
TRigL_TimeOut(CLK:= TimeOut.Q  );

		IF  TRigR_TimeOut.Q THEN     (* Condizione di WARNING *)
					WRN:=TRUE;
 					LogEv(EL_Wrn,EO_PORT,ID,5,'Nessun_Movimento'); (********* Morneo ***********)
		END_IF

		IF  TRigL_TimeOut.Q THEN     (* Condizione di Rientro dal WARNING *)
					WRN:=FALSE;
 					LogEv(EL_Log,EO_PORT,ID,1,'');
		END_IF


(**** Gestione ingresso Analogico per la gestione del valore istantaneo  *****************)

(* Verifico che le variabile letta dall'ingresso Analogico  sia dentro i range
ATTENZIONE I LIMITI SPESSO SONO IN WORD VERIFICA  TABELLA MANUALE WAGO  *)

SegnaleHH:=(AI_INPUT>=SogliaHH);
SegnaleHL:=(AI_INPUT<=SogliaHL);
SegnaleOK:=NOT (SegnaleHH OR SegnaleHL);


(* Linerarizzo il segnale di ingresso e la converto in unita ingegneristiche *)
ValoreScalato:=LINEAR(PuntoMinX, PuntoMaxX, AI_INPUT, PuntoMinY, PuntoMaxY,Decimali);

IF SegnaleOK  THEN
	(*  Verifica  e segnalazione Warning *)
	SegnaleWH:=(ValoreScalato>SogliaWH*(EXPT(10, Decimali)));
	SegnaleWL:=(ValoreScalato<SogliaWL*(EXPT(10, Decimali)));

		FiltroWRN(IN:=(SegnaleWH OR SegnaleWL)  , PT:=INT_TO_TIME(TAP) );    (* Filtro su LOG *)
		IF  FiltroWRN.Q THEN     (* Condizione di WARNING *)
			IF NOT WRN THEN
					WRN:=TRUE;
 					LogEv(EL_Wrn,EO_PORT,ID,SEL(ValoreScalato<=SogliaWL,3,2),INT_TO_STRING(ValoreScalato));
			END_IF
		END_IF


	      IF (INITEV OR WRN OR ERR)  AND NOT FiltroWRN.Q THEN

			FiltroWRN(IN:=FALSE  , PT:=INT_TO_TIME(TAP));    (* Resetto il Filtro su LOG WRN  *)
			FiltroERR(IN:=FALSE  , PT:=INT_TO_TIME(TAP));    (* Resetto il Filtro su LOG ERR *)
			INITEV:=FALSE; ERR:=FALSE; WRN:=FALSE;
			LogEv(EL_Log,EO_PORT,ID,1,'');
		END_IF

		 Status_Vis:=16#20F020;    (* Indicazione WEB Visu Sonda OK *)
ELSE
		FiltroERR(IN:=TRUE  , PT:= INT_TO_TIME(TAP) );    (* Filtro su LOG *)
			IF  FiltroERR.Q THEN     (* Condizione di WARNING *)
					IF NOT ERR THEN
						ERR:=TRUE;
						IF SegnaleHH THEN LogEv(EL_Alarm,EO_PORT,ID,6,INT_TO_STRING(ValoreScalato));END_IF;
						IF SegnaleHL THEN LogEv(EL_Alarm,EO_PORT,ID,4,INT_TO_STRING(ValoreScalato));END_IF;
					END_IF
			END_IF

 		Status_Vis:=16#2020F0;   (* Indicazione WEB Visu Sonda KO *)
		Status_Log:=1;

END_IF
END_FUNCTION_BLOCK

(* POU Plant_Objects/obj_SW_CTB, ST *)
FUNCTION_BLOCK obj_SW_CTB (* Software Energy contabilizer TICK=500ms *)
VAR_INPUT
	(* Settings *)
	ID				: BYTE;
	(* Physical Inputs *)
	T_SEND			: INT; (* 10^-1 °C *)
	T_RET			: INT; (* 10^-1 °C *)
	FLOW			: INT; (* m^3/h *)
END_VAR
VAR_IN_OUT
	(* Persistent counter *)
	ENERGY_WH		: REAL;
	ENERGY			: DWORD; (* 10^-2 MWh *)
END_VAR
VAR_OUTPUT
	POWER_KW		: REAL;
	(* Visu/Log *)
	Status_Log		: BYTE;
	Status_Vis		: DWORD;
END_VAR
VAR
	init			: BOOL;
	overflow		: BOOL;
	P_OLD			: REAL;
END_VAR
(* P0[kW] = FLOW * (8,164 *10 ^ -1 * T_SEND/10 + 9,623*10^2) * 4,186 * (T_SEND - T_RET)/10 / 3600 *)
POWER_KW := ( INT_TO_REAL(FLOW) * ( (8.164E-2 * INT_TO_REAL(T_SEND)) + 9.623E2 ) * 4.1868 * (T_SEND-T_RET) ) / 36000 ;

IF NOT init THEN
	init:=TRUE;
ELSE
	(* E[Wh] = ( (P0+P1)/2 ) * 0,5 / 3600 = (P0+P1)/14400 *)
	ENERGY_WH := ENERGY_WH + (( POWER_KW + P_OLD ) / 14.4);
END_IF

P_OLD:=POWER_KW;

IF ENERGY_WH>10000 THEN
	ENERGY_WH := ENERGY_WH - 10000;
	ENERGY := ENERGY + 1;
END_IF

(* Check status *)
Status_Log:=0; Status_Vis:=16#20F020;
END_FUNCTION_BLOCK

(* POU Plant_Objects/obj_TPV, ST *)
FUNCTION_BLOCK obj_TPV
VAR_INPUT
	(* Settings *)
	ID				: BYTE;
	TAP				: BYTE:=4;	   (* Consecutive checks filter *)
	INITEV			: BOOL:= TRUE; (* Generate init OK event *)
	IN_EMIN			: INT :=-2000; (* Low error limit *)
	IN_WMIN			: INT := -550; (* Low warning value *)
	IN_WMAX			: INT :=  900; (* High warning value *)
	IN_EMAX			: INT := 8500; (* High error limit *)
	ERR_MIN_SHORT	: BOOL:= TRUE; (* TRUE  ==> EMIN=Short        , EMAX=Disconnected
									  FALSE ==> EMIN=Disconnected , EMAX=Short 		 *)
	(* Physical input *)
	IN				: INT;
END_VAR
VAR_OUTPUT
	WRN			: BOOL;	(* Value in warning range *)
	ERR			: BOOL;	(* Value error *)
	HI			: INT;	(* Highest value - cleared by Stat_Reset() action *)
	AVG			: INT; 	(* Average value - updated by Mean() action, cleared by Mean_Reset() action *)
	LOW			: INT;	(* Lowest value  - cleared by Stat_Reset() action *)
END_VAR
VAR
	cnt			: BYTE;
	asum		: DINT;
	acnt		: WORD;
END_VAR
(* Check probe value limits *)
IF IN<=IN_EMIN OR IN>=IN_EMAX THEN
	IF NOT ERR THEN
		cnt:=cnt+1;
		IF cnt>TAP THEN
			cnt:=0;
			ERR:=TRUE; WRN:=FALSE;
			IF ( ERR_MIN_SHORT=TRUE  AND IN<=IN_EMIN ) OR ( ERR_MIN_SHORT=FALSE AND IN>=IN_EMAX ) THEN
				LogEv(EL_Alarm,EO_TPV,ID,5,INT_TO_STRING(IN));
			ELSE
				LogEv(EL_Alarm,EO_TPV,ID,4,INT_TO_STRING(IN));
			END_IF
		END_IF
	END_IF
ELSIF IN<=IN_WMIN OR IN>=IN_WMAX THEN
	IF NOT WRN THEN
		cnt:=cnt+1;
		IF cnt>TAP THEN
			cnt:=0;
			ERR:=FALSE; WRN:=TRUE;
			LogEv(EL_Wrn,EO_TPV,ID,SEL(IN<=IN_WMIN,3,2),INT_TO_STRING(IN));
		END_IF
	END_IF
ELSE
	IF INITEV OR WRN OR ERR THEN
		cnt:=cnt+1;
		IF cnt>TAP THEN
			cnt:=0;
			INITEV:=FALSE; ERR:=FALSE; WRN:=FALSE;
			LogEv(EL_Log,EO_TPV,ID,1,'Probe_OK');
		END_IF
	END_IF
END_IF

(* Average value *)
IF acnt>=60000 THEN
	Mean();
	asum := asum - AVG;
	acnt := acnt - 1;
END_IF

asum := asum + IN;
acnt := acnt + 1;

(* Statistics values *)
IF IN<LOW THEN LOW:=IN; END_IF
IF IN>HI  THEN HI :=IN; END_IF
END_FUNCTION_BLOCK
ACTION Mean:
AVG := DINT_TO_INT(asum/acnt);
END_ACTION
ACTION Mean_Reset:
AVG:=IN;
asum:=IN;
acnt:=1;
END_ACTION
ACTION Stat_Reset:
HI:=IN;
LOW:=IN;
END_ACTION

(* POU Plant_Objects/obj_TPV_SENS, ST *)
FUNCTION_BLOCK obj_TPV_SENS
VAR_INPUT
	(* Settings *)
	ID				: BYTE;
	PuntoMinX		: INT;			(* Parametri per la scalatura *)
	PuntoMaxX		: INT;
	PuntoMinY		: REAL;
	PuntoMaxY		: REAL;
	Decimali		: BYTE;
	SogliaHH		: WORD;			(* Soglia per segnalazione Allarme Extra Range in alto - Solitamente sondo in CC *)
	SogliaHL		: WORD;			(* Soglia per segnalazione Allarme Extra Range in Basso - Solitamente sondo Aperta *)
	SogliaWH		: REAL;			(* Soglia per segnalazione Warning  in alto  *)
	SogliaWL		: REAL;    		(* Soglia per segnalazione Warning in basso  *)
	TAP				: INT:=2000;	(* Filtro in msec *)
	INITEV			: BOOL:= TRUE;	(* Generate init OK event *)

	(* Physical input *)
	AI_INPUT	: WORD;    (* Ingresso Fisico dal modulo Analogico *)

END_VAR
VAR_OUTPUT
	WRN:	BOOL;	(* Segnalazione Warning *)
	ERR: 	BOOL; 	(* Segnalazione Errore *)
	ValoreScalato: INT;
	(* Status *)
	Status_Log	: BYTE;
	Status_Vis 	: DWORD;
END_VAR
VAR

	SegnaleHH: BOOL;
	SegnaleHL: BOOL;
	SegnaleOK: BOOL;

	SegnaleWH: BOOL;
	SegnaleWL: BOOL;

    FiltroWRN:TON;
    FiltroOK:TON;
    FiltroERR:TON;


END_VAR
(* Verifico che le variabile letta dall'ingresso Analogico  sia dentro i range
ATTENZIONE I LIMITI SPESSO SONO IN WORD VERIFICA  TABELLA MANUALE WAGO  *)

SegnaleHH:=(AI_INPUT>=SogliaHH);
SegnaleHL:=(AI_INPUT<=SogliaHL);
SegnaleOK:=NOT (SegnaleHH OR SegnaleHL);

(* Linerarizzo il segnale di ingresso e la converto in unita ingegneristiche *)
ValoreScalato:=LINEAR(PuntoMinX,PuntoMaxX,	AI_INPUT,
					  PuntoMinY,PuntoMaxY,	Decimali);


IF SegnaleOK  THEN

(*  Verifica  e segnalazione Warning *)
	SegnaleWH:=(ValoreScalato>SogliaWH*(EXPT(10, Decimali)));
	SegnaleWL:=(ValoreScalato<SogliaWL*(EXPT(10, Decimali)));

		FiltroWRN(IN:=(SegnaleWH OR SegnaleWL)  , PT:=INT_TO_TIME(TAP) );    (* Filtro su LOG *)
		IF  FiltroWRN.Q THEN     (* Condizione di WARNING *)
			IF NOT WRN THEN
					WRN:=TRUE;
 					LogEv(EL_Wrn,EO_TPV,ID,SEL(ValoreScalato<=SogliaWL,3,2),INT_TO_STRING(ValoreScalato));
			END_IF
		END_IF


	    IF (INITEV OR WRN OR ERR) AND NOT FiltroWRN.Q THEN
			FiltroWRN(IN:=FALSE  , PT:=INT_TO_TIME(TAP));    (* Resetto il Filtro su LOG WRN  *)
			FiltroERR(IN:=FALSE  , PT:=INT_TO_TIME(TAP));    (* Resetto il Filtro su LOG ERR *)
			INITEV:=FALSE; ERR:=FALSE; WRN:=FALSE;
			LogEv(EL_Log,EO_TPV,ID,1,'');
		END_IF

		 Status_Vis:=16#20F020;    (* Indicazione WEB Visu Sonda OK *)
ELSE
		FiltroERR(IN:=TRUE  , PT:= INT_TO_TIME(TAP) );    (* Filtro su LOG *)
			IF  FiltroERR.Q THEN     (* Condizione di WARNING *)
					IF NOT ERR THEN
						ERR:=TRUE;
						IF SegnaleHH THEN LogEv(EL_Alarm,EO_TPV,ID,6,INT_TO_STRING(ValoreScalato));END_IF;
						IF SegnaleHL THEN LogEv(EL_Alarm,EO_TPV,ID,4,INT_TO_STRING(ValoreScalato));END_IF;
					END_IF
			END_IF

 		Status_Vis:=16#2020F0;   (* Indicazione WEB Visu Sonda KO *)

END_IF


(*     Moreno      ********************** Chiedere ad Andrea **

(* Statistics values *)
IF IN<LOW THEN LOW:=IN; END_IF
IF IN>HI  THEN HI :=IN; END_IF
*) 
END_FUNCTION_BLOCK

(* POU PLC_WDT, ST *)
FUNCTION PLC_WDT: DWORD VAR_INPUT dwEvent: DWORD; dwFilter: DWORD; dwOwner: DWORD; END_VAR
LogEv(EL_AlarmStop,EO_SYS,1,10,'Watchdog');
END_FUNCTION

(* POU Utils Functions/RAWTOHEX, ST *)
FUNCTION RAWTOHEX : WORD
VAR_INPUT
	pData: POINTER TO BYTE;
	DataLen: WORD;
	pString: POINTER TO BYTE;
END_VAR
VAR
	xl: WORD;
END_VAR
xl:=0;

WHILE DataLen>0 DO

	pString^ := (pData^ / 16#10) + 48 + (((pData^ / 16#10)/10)*7);
	pString:=pString+1;
	pString^ := (pData^ AND 16#0F)  + 48 + (((pData^ AND 16#0F)/10)*7);
	pString:=pString+1;
	pData:=pData+1;
	DataLen:=DataLen-1;
	xl:=xl+2;

END_WHILE

(*pString^:=0;*)

RAWTOHEX:=xl;
END_FUNCTION

(* POU Utils Functions/RAWTOHEXSTR, ST *)
FUNCTION RAWTOHEXSTR : STRING(128)
VAR_INPUT
	pData: POINTER TO BYTE;
	DataLen: BYTE;
END_VAR
VAR
	pt: POINTER TO BYTE;
	xl: BYTE;
END_VAR
pt:=ADR(RAWTOHEXSTR);

xl:=2;

WHILE DataLen>0 AND xl<128 DO

	pt^ := (pData^ / 16#10) + 48 + (((pData^ / 16#10)/10)*7);
	pt:=pt+1;
	pt^ := (pData^ AND 16#0F)  + 48 + (((pData^ AND 16#0F)/10)*7);
	pt:=pt+1;

	xl:=xl+2;

	DataLen:=DataLen-1;
	pData:=pData+1;

END_WHILE

pt^:=0;
END_FUNCTION

(* POU Utils/RTC_Update, ST *)
FUNCTION RTC_Update : BOOL
VAR
	T: DT;
	TS: STRING;
	TS2: STRING;
	Hour: BYTE;
	Minute: BYTE;
END_VAR
(* Get RTC time *)
T:=SysRtcGetTime(TRUE);
Sys.Time_CT_DT:=T;
(* Calculate variables *)
TS:=DT_TO_STRING(T);
Sys.Time_LogString:=DELETE(STR:=TS, LEN:=3, POS:=1);
TS2:=MID(STR:=TS, LEN:=4, POS:= 4); Sys.Time_Year 	:=STRING_TO_WORD(TS2);
TS2:=MID(STR:=TS, LEN:=2, POS:= 9); Sys.Time_Month	:=STRING_TO_BYTE(TS2);
TS2:=MID(STR:=TS, LEN:=2, POS:=12); Sys.Time_Day  	:=STRING_TO_BYTE(TS2);
Sys.Time_CT_Day:=(32*(Sys.Time_Month-1)+Sys.Time_Day-1);
TS2:=MID(STR:=TS, LEN:=2, POS:=15); Hour			:=STRING_TO_BYTE(TS2);
TS2:=MID(STR:=TS, LEN:=2, POS:=18); Minute		 	:=STRING_TO_BYTE(TS2);
Sys.Time_CT_Quarter:=Hour*4+(Minute/15);
END_FUNCTION

(* Visualisation PLC_VISU
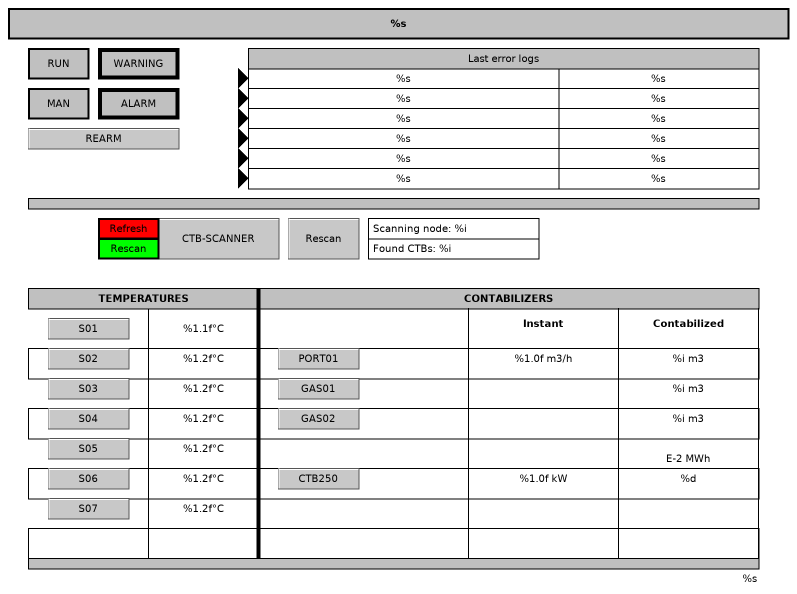
button at (50,350)-(131,371): text "S02"
rectangle at (520,570)-(761,591): text "%s"; shows Sys.Time_LogString
rectangle at (10,10)-(791,41): text "%s"; shows .Plant_NAME
rectangle at (160,350)-(251,371): text "%1.2f°C"; shows INT_TO_REAL(.TPV02.ValoreScalato)/(.TPV02.Decimali*10)
rounded rectangle at (30,50)-(91,81): text "RUN"; alarm colour if NOT Mode_Manual; runs INTERN ASSIGN Mode_Manual:=(FALSE)
rounded rectangle at (30,90)-(91,121): text "MAN"; alarm colour if Mode_Manual; runs INTERN ASSIGN Mode_Manual:=(TRUE)
button at (160,220)-(281,261): text "CTB-SCANNER"; opens VIS_CTBSCAN01
rectangle at (100,90)-(181,121): text "ALARM"; alarm colour if Sys.Alarm; runs INTERN ASSIGN Mode_Manual:=(FALSE)
rectangle at (100,50)-(181,81): text "WARNING"; alarm colour if Sys.Warning; runs INTERN ASSIGN Mode_Manual:=(TRUE)
button at (30,130)-(181,151): text "REARM"; runs INTERN ASSIGN Sys.Alarm:=(FALSE);INTERN ASSIGN Sys.Warning:=(FALSE)
button at (50,320)-(131,341): text "S01"
rectangle at (160,320)-(251,341): text "%1.1f°C"; shows INT_TO_REAL(.TPV01.IN)/10
button at (50,380)-(131,401): text "S03"
rectangle at (160,380)-(251,401): text "%1.2f°C"; shows INT_TO_REAL(.TPV03.ValoreScalato)/(.TPV03.Decimali*10)
button at (50,410)-(131,431): text "S04"
rectangle at (160,410)-(251,431): text "%1.2f°C"; shows INT_TO_REAL(.TPV04.ValoreScalato)/(.TPV04.Decimali*10)
button at (50,440)-(131,461): text "S05"
rectangle at (160,440)-(251,461): text "%1.2f°C"; shows INT_TO_REAL(.TPV05.ValoreScalato)/(.TPV05.Decimali*10)
button at (50,470)-(131,491): text "S06"
rectangle at (160,470)-(251,491): text "%1.2f°C"; shows INT_TO_REAL(.TPV06.ValoreScalato)/(.TPV06.Decimali*10)
button at (50,500)-(131,521): text "S07"
rectangle at (160,500)-(251,521): text "%1.2f°C"; shows INT_TO_REAL(.TPV07.ValoreScalato)/(.TPV07.Decimali*10)
rectangle at (30,290)-(261,311): text "TEMPERATURES"
rectangle at (260,290)-(761,311): text "CONTABILIZERS"
button at (280,350)-(361,371): text "PORT01"
rectangle at (480,350)-(611,371): text "%1.0f m3/h"; shows INT_TO_REAL(.PORT01.ValoreScalato)
rectangle at (470,310)-(621,341): text "Instant"
rectangle at (630,350)-(751,371): text "%i m3"; shows .PortataTotalePORT01
rectangle at (620,310)-(761,341): text "Contabilized"
button at (280,380)-(361,401): text "GAS01"
button at (280,410)-(361,431): text "GAS02"
rectangle at (630,380)-(751,401): text "%i m3"; shows .PortataTotaleGAS01
rectangle at (630,410)-(751,431): text "%i m3"; shows .PortataTotaleGAS02
rectangle at (560,70)-(761,91): text "%s"; shows Sys.LastLogs_Msg[0]
polygon at (240,170)-(250,190): invisible if Sys.LastLogs_Idx<>0
rectangle at (560,90)-(761,111): text "%s"; shows Sys.LastLogs_Msg[1]
polygon at (240,70)-(250,90): invisible if Sys.LastLogs_Idx<>1
rectangle at (560,110)-(761,131): text "%s"; shows Sys.LastLogs_Msg[2]
polygon at (240,90)-(250,110): invisible if Sys.LastLogs_Idx<>2
rectangle at (560,130)-(761,151): text "%s"; shows Sys.LastLogs_Msg[3]
polygon at (240,110)-(250,130): invisible if Sys.LastLogs_Idx<>3
rectangle at (560,150)-(761,171): text "%s"; shows Sys.LastLogs_Msg[4]
polygon at (240,130)-(250,150): invisible if Sys.LastLogs_Idx<>4
rectangle at (560,170)-(761,191): text "%s"; shows Sys.LastLogs_Msg[5]
polygon at (240,150)-(250,170): invisible if Sys.LastLogs_Idx<>5
rectangle at (250,70)-(561,91): text "%s"; shows Sys.LastLogs_Dat[0]
rectangle at (250,90)-(561,111): text "%s"; shows Sys.LastLogs_Dat[1]
rectangle at (250,110)-(561,131): text "%s"; shows Sys.LastLogs_Dat[2]
rectangle at (250,130)-(561,151): text "%s"; shows Sys.LastLogs_Dat[3]
rectangle at (250,150)-(561,171): text "%s"; shows Sys.LastLogs_Dat[4]
rectangle at (250,170)-(561,191): text "%s"; shows Sys.LastLogs_Dat[5]
rectangle at (250,50)-(761,71): text "Last error logs"
button at (290,220)-(361,261): text "Rescan"; runs INTERN ASSIGN CTBSCAN01.Rescan:=(TRUE)
rectangle at (100,220)-(161,241): text "Refresh"; alarm colour if .CTBSCAN01.Refresh
rectangle at (100,240)-(161,261): text "Rescan"; alarm colour if .CTBSCAN01.Rescan
rectangle at (370,240)-(541,261): text "Found CTBs: %i"; shows .CTBSCAN01.ConnectedCTBs
rectangle at (370,220)-(541,241): text "Scanning node: %i"; shows .CTBSCAN01.cnt
rectangle at (480,470)-(611,491): text "%1.0f kW"; shows .CTB250.POWER_KW
rectangle at (630,470)-(751,491): text "%d"; shows .CTB250.ENERGY
button at (280,470)-(361,491): text "CTB250"
rectangle at (630,450)-(751,471): text "E-2 MWh"
11 more shapes without text or variables
13 elements of other kinds (tables, trends, ...) not read
*)

(* Visualisation VIS_CTBSCAN01
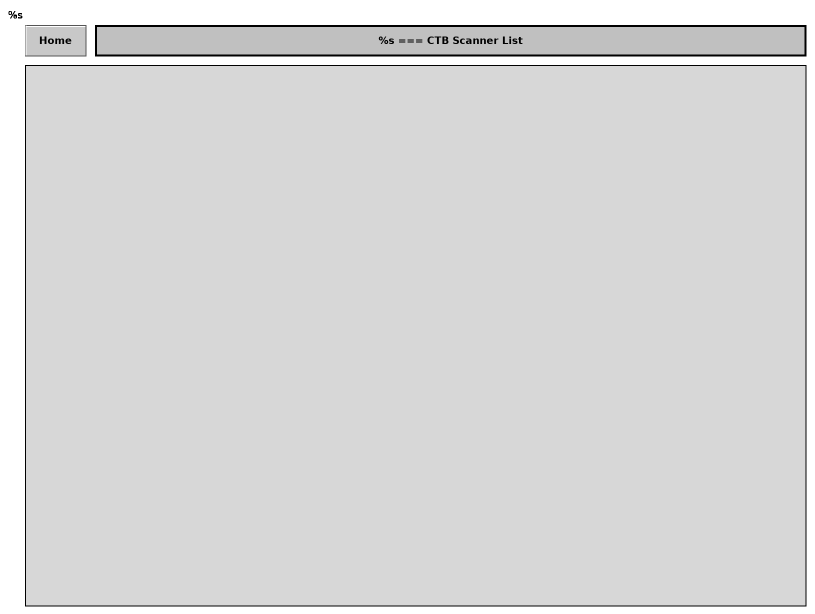
rectangle at (0,0)-(0,0): text "%s"; shows CTBSCAN01.VisuDatiMbus[INDEX].sdNodoPresente; alarm colour if CTBSCAN01.NodoMBusPresente[INDEX]; editable
rectangle at (0,0)-(0,0): text "%s"; shows CTBSCAN01.VisuDatiMbus[INDEX].sdEnergia
rectangle at (0,0)-(0,0): text "%s"; shows CTBSCAN01.VisuDatiMbus[INDEX].sdPotenza
rectangle at (0,0)-(0,0): text "%s"; shows CTBSCAN01.VisuDatiMbus[INDEX].sdVolume
rectangle at (0,0)-(0,0): text "%s"; shows CTBSCAN01.VisuDatiMbus[INDEX].sdFlow
rectangle at (0,0)-(0,0): text "%s"; shows CTBSCAN01.VisuDatiMbus[INDEX].sdTempIngresso
rectangle at (0,0)-(0,0): text "%s"; shows CTBSCAN01.VisuDatiMbus[INDEX].sdTempaUscita
rectangle at (0,0)-(0,0): text "%s"; shows CTBSCAN01.VisuDatiMbus[INDEX].sdTempDelta
rectangle at (80,10)-(791,41): text "%s === CTB Scanner List"; shows .Plant_NAME
button at (10,10)-(71,41): text "Home"; opens PLC_VISU
1 more shapes without text or variables
*)
